Fanuc TP program (LS listing): FM194002.ls

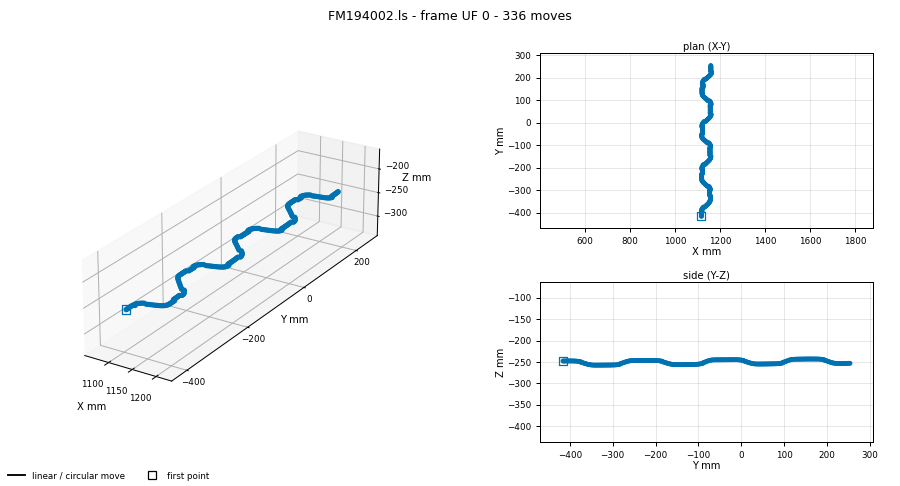
[picture p0: tool path of FM194002.ls in frame UF 0, 336 of 336 moves have a stored position in this frame; points joined in program order, loops and branches not executed]
/PROG  FM194002
/ATTR
OWNER		= MNEDITOR;
COMMENT		= "Auto FANUC move";
PROG_SIZE	= 0;
CREATE		= DATE 26-04-24  TIME 19:40:02;
MODIFIED	= DATE 26-04-24  TIME 19:40:02;
FILE_NAME	= ;
VERSION		= 0;
LINE_COUNT	= 341;
MEMORY_SIZE	= 0;
PROTECT		= READ_WRITE;
TCD:  STACK_SIZE	= 0,
      TASK_PRIORITY	= 50,
      TIME_SLICE	= 0,
      BUSY_LAMP_OFF	= 0,
      ABORT_REQUEST	= 0,
      PAUSE_REQUEST	= 0;
DEFAULT_GROUP	= 1,*,*,*,*;
CONTROL_CODE	= 00000000 00000000;
/MN
   1:  UFRAME_NUM=0 ;
   2:  UTOOL_NUM=1 ;
   3:  R[93]=10 ;
   4:  L P[1] 7mm/sec FINE ;
   5:  L P[2] 7mm/sec FINE ;
   6:  L P[3] 7mm/sec FINE ;
   7:  L P[4] 7mm/sec FINE ;
   8:  L P[5] 7mm/sec FINE ;
   9:  L P[6] 7mm/sec FINE ;
  10:  L P[7] 7mm/sec FINE ;
  11:  L P[8] 7mm/sec FINE ;
  12:  L P[9] 7mm/sec FINE ;
  13:  L P[10] 7mm/sec FINE ;
  14:  L P[11] 7mm/sec FINE ;
  15:  L P[12] 7mm/sec FINE ;
  16:  L P[13] 7mm/sec FINE ;
  17:  L P[14] 7mm/sec FINE ;
  18:  L P[15] 7mm/sec FINE ;
  19:  L P[16] 7mm/sec FINE ;
  20:  L P[17] 7mm/sec FINE ;
  21:  L P[18] 7mm/sec FINE ;
  22:  L P[19] 7mm/sec FINE ;
  23:  L P[20] 7mm/sec FINE ;
  24:  L P[21] 7mm/sec FINE ;
  25:  L P[22] 7mm/sec FINE ;
  26:  L P[23] 7mm/sec FINE ;
  27:  L P[24] 7mm/sec FINE ;
  28:  L P[25] 7mm/sec FINE ;
  29:  L P[26] 7mm/sec FINE ;
  30:  L P[27] 7mm/sec FINE ;
  31:  L P[28] 7mm/sec FINE ;
  32:  L P[29] 7mm/sec FINE ;
  33:  L P[30] 7mm/sec FINE ;
  34:  L P[31] 7mm/sec FINE ;
  35:  L P[32] 7mm/sec FINE ;
  36:  L P[33] 7mm/sec FINE ;
  37:  L P[34] 7mm/sec FINE ;
  38:  L P[35] 7mm/sec FINE ;
  39:  L P[36] 7mm/sec FINE ;
  40:  L P[37] 7mm/sec FINE ;
  41:  L P[38] 7mm/sec FINE ;
  42:  L P[39] 7mm/sec FINE ;
  43:  L P[40] 7mm/sec FINE ;
  44:  L P[41] 7mm/sec FINE ;
  45:  L P[42] 7mm/sec FINE ;
  46:  L P[43] 7mm/sec FINE ;
  47:  L P[44] 7mm/sec FINE ;
  48:  L P[45] 7mm/sec FINE ;
  49:  L P[46] 7mm/sec FINE ;
  50:  L P[47] 7mm/sec FINE ;
  51:  L P[48] 7mm/sec FINE ;
  52:  L P[49] 7mm/sec FINE ;
  53:  L P[50] 7mm/sec FINE ;
  54:  L P[51] 7mm/sec FINE ;
  55:  L P[52] 7mm/sec FINE ;
  56:  L P[53] 7mm/sec FINE ;
  57:  L P[54] 7mm/sec FINE ;
  58:  L P[55] 7mm/sec FINE ;
  59:  L P[56] 7mm/sec FINE ;
  60:  L P[57] 7mm/sec FINE ;
  61:  L P[58] 7mm/sec FINE ;
  62:  L P[59] 7mm/sec FINE ;
  63:  L P[60] 7mm/sec FINE ;
  64:  L P[61] 7mm/sec FINE ;
  65:  L P[62] 7mm/sec FINE ;
  66:  L P[63] 7mm/sec FINE ;
  67:  L P[64] 7mm/sec FINE ;
  68:  L P[65] 7mm/sec FINE ;
  69:  L P[66] 7mm/sec FINE ;
  70:  L P[67] 7mm/sec FINE ;
  71:  L P[68] 7mm/sec FINE ;
  72:  L P[69] 7mm/sec FINE ;
  73:  L P[70] 7mm/sec FINE ;
  74:  L P[71] 7mm/sec FINE ;
  75:  L P[72] 7mm/sec FINE ;
  76:  L P[73] 7mm/sec FINE ;
  77:  L P[74] 7mm/sec FINE ;
  78:  L P[75] 7mm/sec FINE ;
  79:  L P[76] 7mm/sec FINE ;
  80:  L P[77] 7mm/sec FINE ;
  81:  L P[78] 7mm/sec FINE ;
  82:  L P[79] 7mm/sec FINE ;
  83:  L P[80] 7mm/sec FINE ;
  84:  L P[81] 7mm/sec FINE ;
  85:  L P[82] 7mm/sec FINE ;
  86:  L P[83] 7mm/sec FINE ;
  87:  L P[84] 7mm/sec FINE ;
  88:  L P[85] 7mm/sec FINE ;
  89:  L P[86] 7mm/sec FINE ;
  90:  L P[87] 7mm/sec FINE ;
  91:  L P[88] 7mm/sec FINE ;
  92:  L P[89] 7mm/sec FINE ;
  93:  L P[90] 7mm/sec FINE ;
  94:  L P[91] 7mm/sec FINE ;
  95:  L P[92] 7mm/sec FINE ;
  96:  L P[93] 7mm/sec FINE ;
  97:  L P[94] 7mm/sec FINE ;
  98:  L P[95] 7mm/sec FINE ;
  99:  L P[96] 7mm/sec FINE ;
 100:  L P[97] 7mm/sec FINE ;
 101:  L P[98] 7mm/sec FINE ;
 102:  L P[99] 7mm/sec FINE ;
 103:  L P[100] 7mm/sec FINE ;
 104:  L P[101] 7mm/sec FINE ;
 105:  L P[102] 7mm/sec FINE ;
 106:  L P[103] 7mm/sec FINE ;
 107:  L P[104] 7mm/sec FINE ;
 108:  L P[105] 7mm/sec FINE ;
 109:  L P[106] 7mm/sec FINE ;
 110:  L P[107] 7mm/sec FINE ;
 111:  L P[108] 7mm/sec FINE ;
 112:  L P[109] 7mm/sec FINE ;
 113:  L P[110] 7mm/sec FINE ;
 114:  L P[111] 7mm/sec FINE ;
 115:  L P[112] 7mm/sec FINE ;
 116:  L P[113] 7mm/sec FINE ;
 117:  L P[114] 7mm/sec FINE ;
 118:  L P[115] 7mm/sec FINE ;
 119:  L P[116] 7mm/sec FINE ;
 120:  L P[117] 7mm/sec FINE ;
 121:  L P[118] 7mm/sec FINE ;
 122:  L P[119] 7mm/sec FINE ;
 123:  L P[120] 7mm/sec FINE ;
 124:  L P[121] 7mm/sec FINE ;
 125:  L P[122] 7mm/sec FINE ;
 126:  L P[123] 7mm/sec FINE ;
 127:  L P[124] 7mm/sec FINE ;
 128:  L P[125] 7mm/sec FINE ;
 129:  L P[126] 7mm/sec FINE ;
 130:  L P[127] 7mm/sec FINE ;
 131:  L P[128] 7mm/sec FINE ;
 132:  L P[129] 7mm/sec FINE ;
 133:  L P[130] 7mm/sec FINE ;
 134:  L P[131] 7mm/sec FINE ;
 135:  L P[132] 7mm/sec FINE ;
 136:  L P[133] 7mm/sec FINE ;
 137:  L P[134] 7mm/sec FINE ;
 138:  L P[135] 7mm/sec FINE ;
 139:  L P[136] 7mm/sec FINE ;
 140:  L P[137] 7mm/sec FINE ;
 141:  L P[138] 7mm/sec FINE ;
 142:  L P[139] 7mm/sec FINE ;
 143:  L P[140] 7mm/sec FINE ;
 144:  L P[141] 7mm/sec FINE ;
 145:  L P[142] 7mm/sec FINE ;
 146:  L P[143] 7mm/sec FINE ;
 147:  L P[144] 7mm/sec FINE ;
 148:  L P[145] 7mm/sec FINE ;
 149:  L P[146] 7mm/sec FINE ;
 150:  L P[147] 7mm/sec FINE ;
 151:  L P[148] 7mm/sec FINE ;
 152:  L P[149] 7mm/sec FINE ;
 153:  L P[150] 7mm/sec FINE ;
 154:  L P[151] 7mm/sec FINE ;
 155:  L P[152] 7mm/sec FINE ;
 156:  L P[153] 7mm/sec FINE ;
 157:  L P[154] 7mm/sec FINE ;
 158:  L P[155] 7mm/sec FINE ;
 159:  L P[156] 7mm/sec FINE ;
 160:  L P[157] 7mm/sec FINE ;
 161:  L P[158] 7mm/sec FINE ;
 162:  L P[159] 7mm/sec FINE ;
 163:  L P[160] 7mm/sec FINE ;
 164:  L P[161] 7mm/sec FINE ;
 165:  L P[162] 7mm/sec FINE ;
 166:  L P[163] 7mm/sec FINE ;
 167:  L P[164] 7mm/sec FINE ;
 168:  L P[165] 7mm/sec FINE ;
 169:  L P[166] 7mm/sec FINE ;
 170:  L P[167] 7mm/sec FINE ;
 171:  L P[168] 7mm/sec FINE ;
 172:  L P[169] 7mm/sec FINE ;
 173:  L P[170] 7mm/sec FINE ;
 174:  L P[171] 7mm/sec FINE ;
 175:  L P[172] 7mm/sec FINE ;
 176:  L P[173] 7mm/sec FINE ;
 177:  L P[174] 7mm/sec FINE ;
 178:  L P[175] 7mm/sec FINE ;
 179:  L P[176] 7mm/sec FINE ;
 180:  L P[177] 7mm/sec FINE ;
 181:  L P[178] 7mm/sec FINE ;
 182:  L P[179] 7mm/sec FINE ;
 183:  L P[180] 7mm/sec FINE ;
 184:  L P[181] 7mm/sec FINE ;
 185:  L P[182] 7mm/sec FINE ;
 186:  L P[183] 7mm/sec FINE ;
 187:  L P[184] 7mm/sec FINE ;
 188:  L P[185] 7mm/sec FINE ;
 189:  L P[186] 7mm/sec FINE ;
 190:  L P[187] 7mm/sec FINE ;
 191:  L P[188] 7mm/sec FINE ;
 192:  L P[189] 7mm/sec FINE ;
 193:  L P[190] 7mm/sec FINE ;
 194:  L P[191] 7mm/sec FINE ;
 195:  L P[192] 7mm/sec FINE ;
 196:  L P[193] 7mm/sec FINE ;
 197:  L P[194] 7mm/sec FINE ;
 198:  L P[195] 7mm/sec FINE ;
 199:  L P[196] 7mm/sec FINE ;
 200:  L P[197] 7mm/sec FINE ;
 201:  L P[198] 7mm/sec FINE ;
 202:  L P[199] 7mm/sec FINE ;
 203:  L P[200] 7mm/sec FINE ;
 204:  L P[201] 7mm/sec FINE ;
 205:  L P[202] 7mm/sec FINE ;
 206:  L P[203] 7mm/sec FINE ;
 207:  L P[204] 7mm/sec FINE ;
 208:  L P[205] 7mm/sec FINE ;
 209:  L P[206] 7mm/sec FINE ;
 210:  L P[207] 7mm/sec FINE ;
 211:  L P[208] 7mm/sec FINE ;
 212:  L P[209] 7mm/sec FINE ;
 213:  L P[210] 7mm/sec FINE ;
 214:  L P[211] 7mm/sec FINE ;
 215:  L P[212] 7mm/sec FINE ;
 216:  L P[213] 7mm/sec FINE ;
 217:  L P[214] 7mm/sec FINE ;
 218:  L P[215] 7mm/sec FINE ;
 219:  L P[216] 7mm/sec FINE ;
 220:  L P[217] 7mm/sec FINE ;
 221:  L P[218] 7mm/sec FINE ;
 222:  L P[219] 7mm/sec FINE ;
 223:  L P[220] 7mm/sec FINE ;
 224:  L P[221] 7mm/sec FINE ;
 225:  L P[222] 7mm/sec FINE ;
 226:  L P[223] 7mm/sec FINE ;
 227:  L P[224] 7mm/sec FINE ;
 228:  L P[225] 7mm/sec FINE ;
 229:  L P[226] 7mm/sec FINE ;
 230:  L P[227] 7mm/sec FINE ;
 231:  L P[228] 7mm/sec FINE ;
 232:  L P[229] 7mm/sec FINE ;
 233:  L P[230] 7mm/sec FINE ;
 234:  L P[231] 7mm/sec FINE ;
 235:  L P[232] 7mm/sec FINE ;
 236:  L P[233] 7mm/sec FINE ;
 237:  L P[234] 7mm/sec FINE ;
 238:  L P[235] 7mm/sec FINE ;
 239:  L P[236] 7mm/sec FINE ;
 240:  L P[237] 7mm/sec FINE ;
 241:  L P[238] 7mm/sec FINE ;
 242:  L P[239] 7mm/sec FINE ;
 243:  L P[240] 7mm/sec FINE ;
 244:  L P[241] 7mm/sec FINE ;
 245:  L P[242] 7mm/sec FINE ;
 246:  L P[243] 7mm/sec FINE ;
 247:  L P[244] 7mm/sec FINE ;
 248:  L P[245] 7mm/sec FINE ;
 249:  L P[246] 7mm/sec FINE ;
 250:  L P[247] 7mm/sec FINE ;
 251:  L P[248] 7mm/sec FINE ;
 252:  L P[249] 7mm/sec FINE ;
 253:  L P[250] 7mm/sec FINE ;
 254:  L P[251] 7mm/sec FINE ;
 255:  L P[252] 7mm/sec FINE ;
 256:  L P[253] 7mm/sec FINE ;
 257:  L P[254] 7mm/sec FINE ;
 258:  L P[255] 7mm/sec FINE ;
 259:  L P[256] 7mm/sec FINE ;
 260:  L P[257] 7mm/sec FINE ;
 261:  L P[258] 7mm/sec FINE ;
 262:  L P[259] 7mm/sec FINE ;
 263:  L P[260] 7mm/sec FINE ;
 264:  L P[261] 7mm/sec FINE ;
 265:  L P[262] 7mm/sec FINE ;
 266:  L P[263] 7mm/sec FINE ;
 267:  L P[264] 7mm/sec FINE ;
 268:  L P[265] 7mm/sec FINE ;
 269:  L P[266] 7mm/sec FINE ;
 270:  L P[267] 7mm/sec FINE ;
 271:  L P[268] 7mm/sec FINE ;
 272:  L P[269] 7mm/sec FINE ;
 273:  L P[270] 7mm/sec FINE ;
 274:  L P[271] 7mm/sec FINE ;
 275:  L P[272] 7mm/sec FINE ;
 276:  L P[273] 7mm/sec FINE ;
 277:  L P[274] 7mm/sec FINE ;
 278:  L P[275] 7mm/sec FINE ;
 279:  L P[276] 7mm/sec FINE ;
 280:  L P[277] 7mm/sec FINE ;
 281:  L P[278] 7mm/sec FINE ;
 282:  L P[279] 7mm/sec FINE ;
 283:  L P[280] 7mm/sec FINE ;
 284:  L P[281] 7mm/sec FINE ;
 285:  L P[282] 7mm/sec FINE ;
 286:  L P[283] 7mm/sec FINE ;
 287:  L P[284] 7mm/sec FINE ;
 288:  L P[285] 7mm/sec FINE ;
 289:  L P[286] 7mm/sec FINE ;
 290:  L P[287] 7mm/sec FINE ;
 291:  L P[288] 7mm/sec FINE ;
 292:  L P[289] 7mm/sec FINE ;
 293:  L P[290] 7mm/sec FINE ;
 294:  L P[291] 7mm/sec FINE ;
 295:  L P[292] 7mm/sec FINE ;
 296:  L P[293] 7mm/sec FINE ;
 297:  L P[294] 7mm/sec FINE ;
 298:  L P[295] 7mm/sec FINE ;
 299:  L P[296] 7mm/sec FINE ;
 300:  L P[297] 7mm/sec FINE ;
 301:  L P[298] 7mm/sec FINE ;
 302:  L P[299] 7mm/sec FINE ;
 303:  L P[300] 7mm/sec FINE ;
 304:  L P[301] 7mm/sec FINE ;
 305:  L P[302] 7mm/sec FINE ;
 306:  L P[303] 7mm/sec FINE ;
 307:  L P[304] 7mm/sec FINE ;
 308:  L P[305] 7mm/sec FINE ;
 309:  L P[306] 7mm/sec FINE ;
 310:  L P[307] 7mm/sec FINE ;
 311:  L P[308] 7mm/sec FINE ;
 312:  L P[309] 7mm/sec FINE ;
 313:  L P[310] 7mm/sec FINE ;
 314:  L P[311] 7mm/sec FINE ;
 315:  L P[312] 7mm/sec FINE ;
 316:  L P[313] 7mm/sec FINE ;
 317:  L P[314] 7mm/sec FINE ;
 318:  L P[315] 7mm/sec FINE ;
 319:  L P[316] 7mm/sec FINE ;
 320:  L P[317] 7mm/sec FINE ;
 321:  L P[318] 7mm/sec FINE ;
 322:  L P[319] 7mm/sec FINE ;
 323:  L P[320] 7mm/sec FINE ;
 324:  L P[321] 7mm/sec FINE ;
 325:  L P[322] 7mm/sec FINE ;
 326:  L P[323] 7mm/sec FINE ;
 327:  L P[324] 7mm/sec FINE ;
 328:  L P[325] 7mm/sec FINE ;
 329:  L P[326] 7mm/sec FINE ;
 330:  L P[327] 7mm/sec FINE ;
 331:  L P[328] 7mm/sec FINE ;
 332:  L P[329] 7mm/sec FINE ;
 333:  L P[330] 7mm/sec FINE ;
 334:  L P[331] 7mm/sec FINE ;
 335:  L P[332] 7mm/sec FINE ;
 336:  L P[333] 7mm/sec FINE ;
 337:  L P[334] 7mm/sec FINE ;
 338:  L P[335] 7mm/sec FINE ;
 339:  L P[336] 7mm/sec FINE ;
 340:  R[93]=1 ;
 341:  END ;
/POS
P[1]{
   GP1:
	UF : 0, UT : 1,		CONFIG : 'N U T, 0, 0, 0',
	X = 1117.903  mm,	Y = -416.081  mm,	Z = -247.708  mm,
	W = 0.000 deg,	P = 30.000 deg,	R = 175.406 deg
};
P[2]{
   GP1:
	UF : 0, UT : 1,		CONFIG : 'N U T, 0, 0, 0',
	X = 1117.822  mm,	Y = -414.081  mm,	Z = -247.687  mm,
	W = 0.000 deg,	P = 30.000 deg,	R = 175.406 deg
};
P[3]{
   GP1:
	UF : 0, UT : 1,		CONFIG : 'N U T, 0, 0, 0',
	X = 1117.741  mm,	Y = -412.076  mm,	Z = -247.659  mm,
	W = 0.000 deg,	P = 30.000 deg,	R = 175.406 deg
};
P[4]{
   GP1:
	UF : 0, UT : 1,		CONFIG : 'N U T, 0, 0, 0',
	X = 1117.669  mm,	Y = -410.061  mm,	Z = -247.629  mm,
	W = 0.000 deg,	P = 30.000 deg,	R = 175.406 deg
};
P[5]{
   GP1:
	UF : 0, UT : 1,		CONFIG : 'N U T, 0, 0, 0',
	X = 1117.617  mm,	Y = -408.050  mm,	Z = -247.600  mm,
	W = 0.000 deg,	P = 30.000 deg,	R = 175.406 deg
};
P[6]{
   GP1:
	UF : 0, UT : 1,		CONFIG : 'N U T, 0, 0, 0',
	X = 1117.569  mm,	Y = -406.040  mm,	Z = -247.570  mm,
	W = 0.000 deg,	P = 30.000 deg,	R = 175.406 deg
};
P[7]{
   GP1:
	UF : 0, UT : 1,		CONFIG : 'N U T, 0, 0, 0',
	X = 1117.536  mm,	Y = -404.021  mm,	Z = -247.543  mm,
	W = 0.000 deg,	P = 30.000 deg,	R = 175.406 deg
};
P[8]{
   GP1:
	UF : 0, UT : 1,		CONFIG : 'N U T, 0, 0, 0',
	X = 1117.527  mm,	Y = -402.002  mm,	Z = -247.518  mm,
	W = 0.000 deg,	P = 30.000 deg,	R = 175.406 deg
};
P[9]{
   GP1:
	UF : 0, UT : 1,		CONFIG : 'N U T, 0, 0, 0',
	X = 1117.533  mm,	Y = -399.972  mm,	Z = -247.500  mm,
	W = 0.000 deg,	P = 30.000 deg,	R = 175.406 deg
};
P[10]{
   GP1:
	UF : 0, UT : 1,		CONFIG : 'N U T, 0, 0, 0',
	X = 1117.583  mm,	Y = -397.934  mm,	Z = -247.497  mm,
	W = 0.000 deg,	P = 30.000 deg,	R = 175.406 deg
};
P[11]{
   GP1:
	UF : 0, UT : 1,		CONFIG : 'N U T, 0, 0, 0',
	X = 1117.668  mm,	Y = -395.878  mm,	Z = -247.506  mm,
	W = 0.000 deg,	P = 30.000 deg,	R = 175.406 deg
};
P[12]{
   GP1:
	UF : 0, UT : 1,		CONFIG : 'N U T, 0, 0, 0',
	X = 1121.814  mm,	Y = -394.222  mm,	Z = -247.528  mm,
	W = 0.000 deg,	P = 30.000 deg,	R = 175.406 deg
};
P[13]{
   GP1:
	UF : 0, UT : 1,		CONFIG : 'N U T, 0, 0, 0',
	X = 1118.142  mm,	Y = -391.652  mm,	Z = -247.591  mm,
	W = 0.000 deg,	P = 30.000 deg,	R = 169.886 deg
};
P[14]{
   GP1:
	UF : 0, UT : 1,		CONFIG : 'N U T, 0, 0, 0',
	X = 1118.595  mm,	Y = -389.505  mm,	Z = -247.675  mm,
	W = 0.000 deg,	P = 30.000 deg,	R = 162.214 deg
};
P[15]{
   GP1:
	UF : 0, UT : 1,		CONFIG : 'N U T, 0, 0, 0',
	X = 1119.241  mm,	Y = -387.351  mm,	Z = -247.801  mm,
	W = 0.000 deg,	P = 30.000 deg,	R = 154.369 deg
};
P[16]{
   GP1:
	UF : 0, UT : 1,		CONFIG : 'N U T, 0, 0, 0',
	X = 1120.076  mm,	Y = -385.192  mm,	Z = -247.960  mm,
	W = 0.000 deg,	P = 30.000 deg,	R = 146.306 deg
};
P[17]{
   GP1:
	UF : 0, UT : 1,		CONFIG : 'N U T, 0, 0, 0',
	X = 1121.155  mm,	Y = -383.023  mm,	Z = -248.138  mm,
	W = 0.000 deg,	P = 30.000 deg,	R = 137.902 deg
};
P[18]{
   GP1:
	UF : 0, UT : 1,		CONFIG : 'N U T, 0, 0, 0',
	X = 1122.476  mm,	Y = -380.896  mm,	Z = -248.389  mm,
	W = 0.000 deg,	P = 30.000 deg,	R = 137.902 deg
};
P[19]{
   GP1:
	UF : 0, UT : 1,		CONFIG : 'N U T, 0, 0, 0',
	X = 1123.929  mm,	Y = -378.824  mm,	Z = -248.707  mm,
	W = 0.000 deg,	P = 30.000 deg,	R = 137.902 deg
};
P[20]{
   GP1:
	UF : 0, UT : 1,		CONFIG : 'N U T, 0, 0, 0',
	X = 1125.487  mm,	Y = -376.754  mm,	Z = -249.062  mm,
	W = 0.000 deg,	P = 30.000 deg,	R = 137.902 deg
};
P[21]{
   GP1:
	UF : 0, UT : 1,		CONFIG : 'N U T, 0, 0, 0',
	X = 1127.242  mm,	Y = -374.667  mm,	Z = -249.504  mm,
	W = 0.000 deg,	P = 30.000 deg,	R = 137.902 deg
};
P[22]{
   GP1:
	UF : 0, UT : 1,		CONFIG : 'N U T, 0, 0, 0',
	X = 1132.067  mm,	Y = -375.388  mm,	Z = -250.027  mm,
	W = 0.000 deg,	P = 30.000 deg,	R = 137.902 deg
};
P[23]{
   GP1:
	UF : 0, UT : 1,		CONFIG : 'N U T, 0, 0, 0',
	X = 1134.024  mm,	Y = -373.390  mm,	Z = -250.598  mm,
	W = 0.000 deg,	P = 30.000 deg,	R = 137.902 deg
};
P[24]{
   GP1:
	UF : 0, UT : 1,		CONFIG : 'N U T, 0, 0, 0',
	X = 1135.917  mm,	Y = -371.406  mm,	Z = -251.204  mm,
	W = 0.000 deg,	P = 30.000 deg,	R = 137.902 deg
};
P[25]{
   GP1:
	UF : 0, UT : 1,		CONFIG : 'N U T, 0, 0, 0',
	X = 1137.928  mm,	Y = -369.443  mm,	Z = -251.855  mm,
	W = 0.000 deg,	P = 30.000 deg,	R = 137.902 deg
};
P[26]{
   GP1:
	UF : 0, UT : 1,		CONFIG : 'N U T, 0, 0, 0',
	X = 1140.023  mm,	Y = -367.467  mm,	Z = -252.522  mm,
	W = 0.000 deg,	P = 30.000 deg,	R = 137.902 deg
};
P[27]{
   GP1:
	UF : 0, UT : 1,		CONFIG : 'N U T, 0, 0, 0',
	X = 1142.218  mm,	Y = -365.469  mm,	Z = -253.201  mm,
	W = 0.000 deg,	P = 30.000 deg,	R = 137.902 deg
};
P[28]{
   GP1:
	UF : 0, UT : 1,		CONFIG : 'N U T, 0, 0, 0',
	X = 1144.405  mm,	Y = -363.418  mm,	Z = -253.848  mm,
	W = 0.000 deg,	P = 30.000 deg,	R = 137.902 deg
};
P[29]{
   GP1:
	UF : 0, UT : 1,		CONFIG : 'N U T, 0, 0, 0',
	X = 1146.326  mm,	Y = -361.385  mm,	Z = -254.414  mm,
	W = 0.000 deg,	P = 30.000 deg,	R = 137.902 deg
};
P[30]{
   GP1:
	UF : 0, UT : 1,		CONFIG : 'N U T, 0, 0, 0',
	X = 1148.257  mm,	Y = -359.405  mm,	Z = -254.982  mm,
	W = 0.000 deg,	P = 30.000 deg,	R = 146.247 deg
};
P[31]{
   GP1:
	UF : 0, UT : 1,		CONFIG : 'N U T, 0, 0, 0',
	X = 1150.309  mm,	Y = -357.349  mm,	Z = -255.565  mm,
	W = 0.000 deg,	P = 30.000 deg,	R = 158.379 deg
};
P[32]{
   GP1:
	UF : 0, UT : 1,		CONFIG : 'N U T, 0, 0, 0',
	X = 1152.072  mm,	Y = -355.220  mm,	Z = -256.043  mm,
	W = 0.000 deg,	P = 30.000 deg,	R = 169.473 deg
};
P[33]{
   GP1:
	UF : 0, UT : 1,		CONFIG : 'N U T, 0, 0, 0',
	X = 1153.595  mm,	Y = -353.081  mm,	Z = -256.439  mm,
	W = 0.000 deg,	P = 30.000 deg,	R = 179.925 deg
};
P[34]{
   GP1:
	UF : 0, UT : 1,		CONFIG : 'N U T, 0, 0, 0',
	X = 1154.836  mm,	Y = -350.912  mm,	Z = -256.747  mm,
	W = 0.000 deg,	P = 30.000 deg,	R = 179.925 deg
};
P[35]{
   GP1:
	UF : 0, UT : 1,		CONFIG : 'N U T, 0, 0, 0',
	X = 1155.808  mm,	Y = -348.771  mm,	Z = -256.977  mm,
	W = 0.000 deg,	P = 30.000 deg,	R = 179.925 deg
};
P[36]{
   GP1:
	UF : 0, UT : 1,		CONFIG : 'N U T, 0, 0, 0',
	X = 1156.640  mm,	Y = -346.586  mm,	Z = -257.166  mm,
	W = 0.000 deg,	P = 30.000 deg,	R = 179.925 deg
};
P[37]{
   GP1:
	UF : 0, UT : 1,		CONFIG : 'N U T, 0, 0, 0',
	X = 1157.161  mm,	Y = -344.331  mm,	Z = -257.271  mm,
	W = 0.000 deg,	P = 30.000 deg,	R = 179.925 deg
};
P[38]{
   GP1:
	UF : 0, UT : 1,		CONFIG : 'N U T, 0, 0, 0',
	X = 1157.393  mm,	Y = -342.172  mm,	Z = -257.304  mm,
	W = 0.000 deg,	P = 30.000 deg,	R = 179.925 deg
};
P[39]{
   GP1:
	UF : 0, UT : 1,		CONFIG : 'N U T, 0, 0, 0',
	X = 1157.531  mm,	Y = -340.095  mm,	Z = -257.316  mm,
	W = 0.000 deg,	P = 30.000 deg,	R = 179.925 deg
};
P[40]{
   GP1:
	UF : 0, UT : 1,		CONFIG : 'N U T, 0, 0, 0',
	X = 1157.590  mm,	Y = -338.047  mm,	Z = -257.316  mm,
	W = 0.000 deg,	P = 30.000 deg,	R = 179.925 deg
};
P[41]{
   GP1:
	UF : 0, UT : 1,		CONFIG : 'N U T, 0, 0, 0',
	X = 1157.627  mm,	Y = -336.032  mm,	Z = -257.313  mm,
	W = 0.000 deg,	P = 30.000 deg,	R = 179.925 deg
};
P[42]{
   GP1:
	UF : 0, UT : 1,		CONFIG : 'N U T, 0, 0, 0',
	X = 1157.653  mm,	Y = -334.022  mm,	Z = -257.307  mm,
	W = 0.000 deg,	P = 30.000 deg,	R = 179.925 deg
};
P[43]{
   GP1:
	UF : 0, UT : 1,		CONFIG : 'N U T, 0, 0, 0',
	X = 1157.672  mm,	Y = -332.016  mm,	Z = -257.298  mm,
	W = 0.000 deg,	P = 30.000 deg,	R = 179.925 deg
};
P[44]{
   GP1:
	UF : 0, UT : 1,		CONFIG : 'N U T, 0, 0, 0',
	X = 1157.685  mm,	Y = -330.011  mm,	Z = -257.283  mm,
	W = 0.000 deg,	P = 30.000 deg,	R = 179.925 deg
};
P[45]{
   GP1:
	UF : 0, UT : 1,		CONFIG : 'N U T, 0, 0, 0',
	X = 1157.693  mm,	Y = -328.007  mm,	Z = -257.262  mm,
	W = 0.000 deg,	P = 30.000 deg,	R = 179.925 deg
};
P[46]{
   GP1:
	UF : 0, UT : 1,		CONFIG : 'N U T, 0, 0, 0',
	X = 1157.700  mm,	Y = -326.005  mm,	Z = -257.241  mm,
	W = 0.000 deg,	P = 30.000 deg,	R = 179.925 deg
};
P[47]{
   GP1:
	UF : 0, UT : 1,		CONFIG : 'N U T, 0, 0, 0',
	X = 1157.703  mm,	Y = -324.003  mm,	Z = -257.219  mm,
	W = 0.000 deg,	P = 30.000 deg,	R = 179.925 deg
};
P[48]{
   GP1:
	UF : 0, UT : 1,		CONFIG : 'N U T, 0, 0, 0',
	X = 1153.706  mm,	Y = -321.999  mm,	Z = -257.197  mm,
	W = 0.000 deg,	P = 30.000 deg,	R = 179.925 deg
};
P[49]{
   GP1:
	UF : 0, UT : 1,		CONFIG : 'N U T, 0, 0, 0',
	X = 1153.704  mm,	Y = -320.005  mm,	Z = -257.178  mm,
	W = 0.000 deg,	P = 30.000 deg,	R = 179.925 deg
};
P[50]{
   GP1:
	UF : 0, UT : 1,		CONFIG : 'N U T, 0, 0, 0',
	X = 1153.696  mm,	Y = -318.010  mm,	Z = -257.160  mm,
	W = 0.000 deg,	P = 30.000 deg,	R = 179.925 deg
};
P[51]{
   GP1:
	UF : 0, UT : 1,		CONFIG : 'N U T, 0, 0, 0',
	X = 1153.685  mm,	Y = -316.013  mm,	Z = -257.148  mm,
	W = 0.000 deg,	P = 30.000 deg,	R = 179.925 deg
};
P[52]{
   GP1:
	UF : 0, UT : 1,		CONFIG : 'N U T, 0, 0, 0',
	X = 1153.670  mm,	Y = -314.020  mm,	Z = -257.138  mm,
	W = 0.000 deg,	P = 30.000 deg,	R = 179.925 deg
};
P[53]{
   GP1:
	UF : 0, UT : 1,		CONFIG : 'N U T, 0, 0, 0',
	X = 1153.645  mm,	Y = -312.032  mm,	Z = -257.126  mm,
	W = 0.000 deg,	P = 30.000 deg,	R = 179.925 deg
};
P[54]{
   GP1:
	UF : 0, UT : 1,		CONFIG : 'N U T, 0, 0, 0',
	X = 1153.607  mm,	Y = -310.048  mm,	Z = -257.109  mm,
	W = 0.000 deg,	P = 30.000 deg,	R = 179.925 deg
};
P[55]{
   GP1:
	UF : 0, UT : 1,		CONFIG : 'N U T, 0, 0, 0',
	X = 1153.548  mm,	Y = -308.060  mm,	Z = -257.085  mm,
	W = 0.000 deg,	P = 30.000 deg,	R = 179.925 deg
};
P[56]{
   GP1:
	UF : 0, UT : 1,		CONFIG : 'N U T, 0, 0, 0',
	X = 1153.487  mm,	Y = -306.064  mm,	Z = -257.061  mm,
	W = 0.000 deg,	P = 30.000 deg,	R = 179.925 deg
};
P[57]{
   GP1:
	UF : 0, UT : 1,		CONFIG : 'N U T, 0, 0, 0',
	X = 1153.420  mm,	Y = -304.075  mm,	Z = -257.035  mm,
	W = 0.000 deg,	P = 30.000 deg,	R = 179.925 deg
};
P[58]{
   GP1:
	UF : 0, UT : 1,		CONFIG : 'N U T, 0, 0, 0',
	X = 1153.338  mm,	Y = -302.094  mm,	Z = -257.001  mm,
	W = 0.000 deg,	P = 30.000 deg,	R = 179.925 deg
};
P[59]{
   GP1:
	UF : 0, UT : 1,		CONFIG : 'N U T, 0, 0, 0',
	X = 1157.227  mm,	Y = -299.889  mm,	Z = -256.960  mm,
	W = 0.000 deg,	P = 30.000 deg,	R = -172.261 deg
};
P[60]{
   GP1:
	UF : 0, UT : 1,		CONFIG : 'N U T, 0, 0, 0',
	X = 1157.108  mm,	Y = -297.863  mm,	Z = -256.914  mm,
	W = 0.000 deg,	P = 30.000 deg,	R = -163.648 deg
};
P[61]{
   GP1:
	UF : 0, UT : 1,		CONFIG : 'N U T, 0, 0, 0',
	X = 1156.941  mm,	Y = -295.770  mm,	Z = -256.860  mm,
	W = 0.000 deg,	P = 30.000 deg,	R = -155.021 deg
};
P[62]{
   GP1:
	UF : 0, UT : 1,		CONFIG : 'N U T, 0, 0, 0',
	X = 1156.585  mm,	Y = -293.494  mm,	Z = -256.766  mm,
	W = 0.000 deg,	P = 30.000 deg,	R = -146.317 deg
};
P[63]{
   GP1:
	UF : 0, UT : 1,		CONFIG : 'N U T, 0, 0, 0',
	X = 1155.778  mm,	Y = -291.291  mm,	Z = -256.533  mm,
	W = 0.000 deg,	P = 30.000 deg,	R = -137.092 deg
};
P[64]{
   GP1:
	UF : 0, UT : 1,		CONFIG : 'N U T, 0, 0, 0',
	X = 1154.940  mm,	Y = -289.140  mm,	Z = -256.291  mm,
	W = 0.000 deg,	P = 30.000 deg,	R = -137.092 deg
};
P[65]{
   GP1:
	UF : 0, UT : 1,		CONFIG : 'N U T, 0, 0, 0',
	X = 1153.690  mm,	Y = -286.928  mm,	Z = -255.943  mm,
	W = 0.000 deg,	P = 30.000 deg,	R = -137.092 deg
};
P[66]{
   GP1:
	UF : 0, UT : 1,		CONFIG : 'N U T, 0, 0, 0',
	X = 1152.204  mm,	Y = -284.813  mm,	Z = -255.513  mm,
	W = 0.000 deg,	P = 30.000 deg,	R = -137.092 deg
};
P[67]{
   GP1:
	UF : 0, UT : 1,		CONFIG : 'N U T, 0, 0, 0',
	X = 1150.545  mm,	Y = -282.671  mm,	Z = -255.041  mm,
	W = 0.000 deg,	P = 30.000 deg,	R = -137.092 deg
};
P[68]{
   GP1:
	UF : 0, UT : 1,		CONFIG : 'N U T, 0, 0, 0',
	X = 1145.642  mm,	Y = -283.430  mm,	Z = -254.415  mm,
	W = 0.000 deg,	P = 30.000 deg,	R = -137.092 deg
};
P[69]{
   GP1:
	UF : 0, UT : 1,		CONFIG : 'N U T, 0, 0, 0',
	X = 1143.569  mm,	Y = -281.439  mm,	Z = -253.764  mm,
	W = 0.000 deg,	P = 30.000 deg,	R = -137.092 deg
};
P[70]{
   GP1:
	UF : 0, UT : 1,		CONFIG : 'N U T, 0, 0, 0',
	X = 1141.558  mm,	Y = -279.486  mm,	Z = -253.115  mm,
	W = 0.000 deg,	P = 30.000 deg,	R = -137.092 deg
};
P[71]{
   GP1:
	UF : 0, UT : 1,		CONFIG : 'N U T, 0, 0, 0',
	X = 1139.168  mm,	Y = -277.477  mm,	Z = -252.354  mm,
	W = 0.000 deg,	P = 30.000 deg,	R = -137.092 deg
};
P[72]{
   GP1:
	UF : 0, UT : 1,		CONFIG : 'N U T, 0, 0, 0',
	X = 1137.118  mm,	Y = -275.431  mm,	Z = -251.708  mm,
	W = 0.000 deg,	P = 30.000 deg,	R = -137.092 deg
};
P[73]{
   GP1:
	UF : 0, UT : 1,		CONFIG : 'N U T, 0, 0, 0',
	X = 1135.038  mm,	Y = -273.445  mm,	Z = -251.008  mm,
	W = 0.000 deg,	P = 30.000 deg,	R = -137.092 deg
};
P[74]{
   GP1:
	UF : 0, UT : 1,		CONFIG : 'N U T, 0, 0, 0',
	X = 1132.925  mm,	Y = -271.417  mm,	Z = -250.292  mm,
	W = 0.000 deg,	P = 30.000 deg,	R = -137.092 deg
};
P[75]{
   GP1:
	UF : 0, UT : 1,		CONFIG : 'N U T, 0, 0, 0',
	X = 1131.034  mm,	Y = -269.457  mm,	Z = -249.652  mm,
	W = 0.000 deg,	P = 30.000 deg,	R = -137.092 deg
};
P[76]{
   GP1:
	UF : 0, UT : 1,		CONFIG : 'N U T, 0, 0, 0',
	X = 1128.718  mm,	Y = -267.465  mm,	Z = -248.952  mm,
	W = 0.000 deg,	P = 30.000 deg,	R = -144.940 deg
};
P[77]{
   GP1:
	UF : 0, UT : 1,		CONFIG : 'N U T, 0, 0, 0',
	X = 1126.623  mm,	Y = -265.346  mm,	Z = -248.378  mm,
	W = 0.000 deg,	P = 30.000 deg,	R = -157.359 deg
};
P[78]{
   GP1:
	UF : 0, UT : 1,		CONFIG : 'N U T, 0, 0, 0',
	X = 1124.911  mm,	Y = -263.289  mm,	Z = -247.921  mm,
	W = 0.000 deg,	P = 30.000 deg,	R = -168.781 deg
};
P[79]{
   GP1:
	UF : 0, UT : 1,		CONFIG : 'N U T, 0, 0, 0',
	X = 1123.138  mm,	Y = -261.212  mm,	Z = -247.447  mm,
	W = 0.000 deg,	P = 30.000 deg,	R = 179.652 deg
};
P[80]{
   GP1:
	UF : 0, UT : 1,		CONFIG : 'N U T, 0, 0, 0',
	X = 1121.702  mm,	Y = -259.072  mm,	Z = -247.117  mm,
	W = 0.000 deg,	P = 30.000 deg,	R = 179.652 deg
};
P[81]{
   GP1:
	UF : 0, UT : 1,		CONFIG : 'N U T, 0, 0, 0',
	X = 1120.407  mm,	Y = -256.906  mm,	Z = -246.842  mm,
	W = 0.000 deg,	P = 30.000 deg,	R = 179.652 deg
};
P[82]{
   GP1:
	UF : 0, UT : 1,		CONFIG : 'N U T, 0, 0, 0',
	X = 1119.423  mm,	Y = -254.501  mm,	Z = -246.659  mm,
	W = 0.000 deg,	P = 30.000 deg,	R = 179.652 deg
};
P[83]{
   GP1:
	UF : 0, UT : 1,		CONFIG : 'N U T, 0, 0, 0',
	X = 1119.162  mm,	Y = -252.164  mm,	Z = -246.603  mm,
	W = 0.000 deg,	P = 30.000 deg,	R = 179.652 deg
};
P[84]{
   GP1:
	UF : 0, UT : 1,		CONFIG : 'N U T, 0, 0, 0',
	X = 1119.033  mm,	Y = -250.103  mm,	Z = -246.560  mm,
	W = 0.000 deg,	P = 30.000 deg,	R = 179.652 deg
};
P[85]{
   GP1:
	UF : 0, UT : 1,		CONFIG : 'N U T, 0, 0, 0',
	X = 1118.950  mm,	Y = -248.057  mm,	Z = -246.519  mm,
	W = 0.000 deg,	P = 30.000 deg,	R = 179.652 deg
};
P[86]{
   GP1:
	UF : 0, UT : 1,		CONFIG : 'N U T, 0, 0, 0',
	X = 1118.916  mm,	Y = -246.021  mm,	Z = -246.492  mm,
	W = 0.000 deg,	P = 30.000 deg,	R = 179.652 deg
};
P[87]{
   GP1:
	UF : 0, UT : 1,		CONFIG : 'N U T, 0, 0, 0',
	X = 1118.906  mm,	Y = -244.003  mm,	Z = -246.468  mm,
	W = 0.000 deg,	P = 30.000 deg,	R = 179.652 deg
};
P[88]{
   GP1:
	UF : 0, UT : 1,		CONFIG : 'N U T, 0, 0, 0',
	X = 1118.910  mm,	Y = -241.997  mm,	Z = -246.451  mm,
	W = 0.000 deg,	P = 30.000 deg,	R = 179.652 deg
};
P[89]{
   GP1:
	UF : 0, UT : 1,		CONFIG : 'N U T, 0, 0, 0',
	X = 1118.913  mm,	Y = -239.996  mm,	Z = -246.434  mm,
	W = 0.000 deg,	P = 30.000 deg,	R = 179.652 deg
};
P[90]{
   GP1:
	UF : 0, UT : 1,		CONFIG : 'N U T, 0, 0, 0',
	X = 1118.917  mm,	Y = -237.995  mm,	Z = -246.415  mm,
	W = 0.000 deg,	P = 30.000 deg,	R = 179.652 deg
};
P[91]{
   GP1:
	UF : 0, UT : 1,		CONFIG : 'N U T, 0, 0, 0',
	X = 1118.923  mm,	Y = -235.994  mm,	Z = -246.394  mm,
	W = 0.000 deg,	P = 30.000 deg,	R = 179.652 deg
};
P[92]{
   GP1:
	UF : 0, UT : 1,		CONFIG : 'N U T, 0, 0, 0',
	X = 1118.929  mm,	Y = -233.993  mm,	Z = -246.378  mm,
	W = 0.000 deg,	P = 30.000 deg,	R = 179.652 deg
};
P[93]{
   GP1:
	UF : 0, UT : 1,		CONFIG : 'N U T, 0, 0, 0',
	X = 1118.936  mm,	Y = -231.993  mm,	Z = -246.364  mm,
	W = 0.000 deg,	P = 30.000 deg,	R = 179.652 deg
};
P[94]{
   GP1:
	UF : 0, UT : 1,		CONFIG : 'N U T, 0, 0, 0',
	X = 1118.942  mm,	Y = -229.994  mm,	Z = -246.348  mm,
	W = 0.000 deg,	P = 30.000 deg,	R = 179.652 deg
};
P[95]{
   GP1:
	UF : 0, UT : 1,		CONFIG : 'N U T, 0, 0, 0',
	X = 1118.948  mm,	Y = -227.990  mm,	Z = -246.333  mm,
	W = 0.000 deg,	P = 30.000 deg,	R = 179.652 deg
};
P[96]{
   GP1:
	UF : 0, UT : 1,		CONFIG : 'N U T, 0, 0, 0',
	X = 1122.962  mm,	Y = -226.020  mm,	Z = -246.316  mm,
	W = 0.000 deg,	P = 30.000 deg,	R = 179.652 deg
};
P[97]{
   GP1:
	UF : 0, UT : 1,		CONFIG : 'N U T, 0, 0, 0',
	X = 1122.987  mm,	Y = -224.026  mm,	Z = -246.304  mm,
	W = 0.000 deg,	P = 30.000 deg,	R = 179.652 deg
};
P[98]{
   GP1:
	UF : 0, UT : 1,		CONFIG : 'N U T, 0, 0, 0',
	X = 1123.014  mm,	Y = -222.030  mm,	Z = -246.293  mm,
	W = 0.000 deg,	P = 30.000 deg,	R = 179.652 deg
};
P[99]{
   GP1:
	UF : 0, UT : 1,		CONFIG : 'N U T, 0, 0, 0',
	X = 1123.048  mm,	Y = -220.037  mm,	Z = -246.280  mm,
	W = 0.000 deg,	P = 30.000 deg,	R = 179.652 deg
};
P[100]{
   GP1:
	UF : 0, UT : 1,		CONFIG : 'N U T, 0, 0, 0',
	X = 1123.088  mm,	Y = -218.051  mm,	Z = -246.267  mm,
	W = 0.000 deg,	P = 30.000 deg,	R = 179.652 deg
};
P[101]{
   GP1:
	UF : 0, UT : 1,		CONFIG : 'N U T, 0, 0, 0',
	X = 1123.149  mm,	Y = -216.067  mm,	Z = -246.260  mm,
	W = 0.000 deg,	P = 30.000 deg,	R = 179.652 deg
};
P[102]{
   GP1:
	UF : 0, UT : 1,		CONFIG : 'N U T, 0, 0, 0',
	X = 1123.221  mm,	Y = -214.068  mm,	Z = -246.254  mm,
	W = 0.000 deg,	P = 30.000 deg,	R = 179.652 deg
};
P[103]{
   GP1:
	UF : 0, UT : 1,		CONFIG : 'N U T, 0, 0, 0',
	X = 1123.286  mm,	Y = -212.068  mm,	Z = -246.255  mm,
	W = 0.000 deg,	P = 30.000 deg,	R = 179.652 deg
};
P[104]{
   GP1:
	UF : 0, UT : 1,		CONFIG : 'N U T, 0, 0, 0',
	X = 1123.357  mm,	Y = -210.081  mm,	Z = -246.257  mm,
	W = 0.000 deg,	P = 30.000 deg,	R = 179.652 deg
};
P[105]{
   GP1:
	UF : 0, UT : 1,		CONFIG : 'N U T, 0, 0, 0',
	X = 1123.447  mm,	Y = -208.107  mm,	Z = -246.265  mm,
	W = 0.000 deg,	P = 30.000 deg,	R = 179.652 deg
};
P[106]{
   GP1:
	UF : 0, UT : 1,		CONFIG : 'N U T, 0, 0, 0',
	X = 1119.579  mm,	Y = -205.848  mm,	Z = -246.280  mm,
	W = 0.000 deg,	P = 30.000 deg,	R = 172.109 deg
};
P[107]{
   GP1:
	UF : 0, UT : 1,		CONFIG : 'N U T, 0, 0, 0',
	X = 1119.767  mm,	Y = -203.777  mm,	Z = -246.306  mm,
	W = 0.000 deg,	P = 30.000 deg,	R = 163.850 deg
};
P[108]{
   GP1:
	UF : 0, UT : 1,		CONFIG : 'N U T, 0, 0, 0',
	X = 1120.055  mm,	Y = -201.642  mm,	Z = -246.357  mm,
	W = 0.000 deg,	P = 30.000 deg,	R = 155.549 deg
};
P[109]{
   GP1:
	UF : 0, UT : 1,		CONFIG : 'N U T, 0, 0, 0',
	X = 1120.547  mm,	Y = -199.499  mm,	Z = -246.457  mm,
	W = 0.000 deg,	P = 30.000 deg,	R = 147.099 deg
};
P[110]{
   GP1:
	UF : 0, UT : 1,		CONFIG : 'N U T, 0, 0, 0',
	X = 1121.153  mm,	Y = -197.389  mm,	Z = -246.574  mm,
	W = 0.000 deg,	P = 30.000 deg,	R = 138.529 deg
};
P[111]{
   GP1:
	UF : 0, UT : 1,		CONFIG : 'N U T, 0, 0, 0',
	X = 1121.912  mm,	Y = -195.252  mm,	Z = -246.733  mm,
	W = 0.000 deg,	P = 30.000 deg,	R = 138.529 deg
};
P[112]{
   GP1:
	UF : 0, UT : 1,		CONFIG : 'N U T, 0, 0, 0',
	X = 1122.893  mm,	Y = -193.083  mm,	Z = -246.935  mm,
	W = 0.000 deg,	P = 30.000 deg,	R = 138.529 deg
};
P[113]{
   GP1:
	UF : 0, UT : 1,		CONFIG : 'N U T, 0, 0, 0',
	X = 1124.136  mm,	Y = -190.935  mm,	Z = -247.164  mm,
	W = 0.000 deg,	P = 30.000 deg,	R = 138.529 deg
};
P[114]{
   GP1:
	UF : 0, UT : 1,		CONFIG : 'N U T, 0, 0, 0',
	X = 1125.568  mm,	Y = -188.827  mm,	Z = -247.478  mm,
	W = 0.000 deg,	P = 30.000 deg,	R = 138.529 deg
};
P[115]{
   GP1:
	UF : 0, UT : 1,		CONFIG : 'N U T, 0, 0, 0',
	X = 1127.155  mm,	Y = -186.762  mm,	Z = -247.866  mm,
	W = 0.000 deg,	P = 30.000 deg,	R = 138.529 deg
};
P[116]{
   GP1:
	UF : 0, UT : 1,		CONFIG : 'N U T, 0, 0, 0',
	X = 1128.829  mm,	Y = -184.689  mm,	Z = -248.300  mm,
	W = 0.000 deg,	P = 30.000 deg,	R = 138.529 deg
};
P[117]{
   GP1:
	UF : 0, UT : 1,		CONFIG : 'N U T, 0, 0, 0',
	X = 1133.651  mm,	Y = -185.373  mm,	Z = -248.827  mm,
	W = 0.000 deg,	P = 30.000 deg,	R = 138.529 deg
};
P[118]{
   GP1:
	UF : 0, UT : 1,		CONFIG : 'N U T, 0, 0, 0',
	X = 1135.538  mm,	Y = -183.405  mm,	Z = -249.377  mm,
	W = 0.000 deg,	P = 30.000 deg,	R = 138.529 deg
};
P[119]{
   GP1:
	UF : 0, UT : 1,		CONFIG : 'N U T, 0, 0, 0',
	X = 1137.539  mm,	Y = -181.436  mm,	Z = -249.975  mm,
	W = 0.000 deg,	P = 30.000 deg,	R = 138.529 deg
};
P[120]{
   GP1:
	UF : 0, UT : 1,		CONFIG : 'N U T, 0, 0, 0',
	X = 1139.635  mm,	Y = -179.435  mm,	Z = -250.657  mm,
	W = 0.000 deg,	P = 30.000 deg,	R = 138.529 deg
};
P[121]{
   GP1:
	UF : 0, UT : 1,		CONFIG : 'N U T, 0, 0, 0',
	X = 1141.666  mm,	Y = -177.427  mm,	Z = -251.292  mm,
	W = 0.000 deg,	P = 30.000 deg,	R = 138.529 deg
};
P[122]{
   GP1:
	UF : 0, UT : 1,		CONFIG : 'N U T, 0, 0, 0',
	X = 1143.712  mm,	Y = -175.434  mm,	Z = -251.920  mm,
	W = 0.000 deg,	P = 30.000 deg,	R = 138.529 deg
};
P[123]{
   GP1:
	UF : 0, UT : 1,		CONFIG : 'N U T, 0, 0, 0',
	X = 1145.784  mm,	Y = -173.421  mm,	Z = -252.534  mm,
	W = 0.000 deg,	P = 30.000 deg,	R = 143.864 deg
};
P[124]{
   GP1:
	UF : 0, UT : 1,		CONFIG : 'N U T, 0, 0, 0',
	X = 1147.767  mm,	Y = -171.417  mm,	Z = -253.118  mm,
	W = 0.000 deg,	P = 30.000 deg,	R = 155.227 deg
};
P[125]{
   GP1:
	UF : 0, UT : 1,		CONFIG : 'N U T, 0, 0, 0',
	X = 1149.806  mm,	Y = -169.415  mm,	Z = -253.706  mm,
	W = 0.000 deg,	P = 30.000 deg,	R = 166.755 deg
};
P[126]{
   GP1:
	UF : 0, UT : 1,		CONFIG : 'N U T, 0, 0, 0',
	X = 1151.836  mm,	Y = -167.349  mm,	Z = -254.276  mm,
	W = 0.000 deg,	P = 30.000 deg,	R = 178.077 deg
};
P[127]{
   GP1:
	UF : 0, UT : 1,		CONFIG : 'N U T, 0, 0, 0',
	X = 1153.596  mm,	Y = -165.267  mm,	Z = -254.752  mm,
	W = 0.000 deg,	P = 30.000 deg,	R = 178.077 deg
};
P[128]{
   GP1:
	UF : 0, UT : 1,		CONFIG : 'N U T, 0, 0, 0',
	X = 1155.258  mm,	Y = -163.171  mm,	Z = -255.198  mm,
	W = 0.000 deg,	P = 30.000 deg,	R = 178.077 deg
};
P[129]{
   GP1:
	UF : 0, UT : 1,		CONFIG : 'N U T, 0, 0, 0',
	X = 1156.665  mm,	Y = -161.009  mm,	Z = -255.554  mm,
	W = 0.000 deg,	P = 30.000 deg,	R = 178.077 deg
};
P[130]{
   GP1:
	UF : 0, UT : 1,		CONFIG : 'N U T, 0, 0, 0',
	X = 1157.796  mm,	Y = -158.826  mm,	Z = -255.828  mm,
	W = 0.000 deg,	P = 30.000 deg,	R = 178.077 deg
};
P[131]{
   GP1:
	UF : 0, UT : 1,		CONFIG : 'N U T, 0, 0, 0',
	X = 1158.657  mm,	Y = -156.612  mm,	Z = -256.022  mm,
	W = 0.000 deg,	P = 30.000 deg,	R = 178.077 deg
};
P[132]{
   GP1:
	UF : 0, UT : 1,		CONFIG : 'N U T, 0, 0, 0',
	X = 1159.225  mm,	Y = -154.375  mm,	Z = -256.144  mm,
	W = 0.000 deg,	P = 30.000 deg,	R = 178.077 deg
};
P[133]{
   GP1:
	UF : 0, UT : 1,		CONFIG : 'N U T, 0, 0, 0',
	X = 1159.504  mm,	Y = -152.218  mm,	Z = -256.190  mm,
	W = 0.000 deg,	P = 30.000 deg,	R = 178.077 deg
};
P[134]{
   GP1:
	UF : 0, UT : 1,		CONFIG : 'N U T, 0, 0, 0',
	X = 1159.694  mm,	Y = -150.137  mm,	Z = -256.215  mm,
	W = 0.000 deg,	P = 30.000 deg,	R = 178.077 deg
};
P[135]{
   GP1:
	UF : 0, UT : 1,		CONFIG : 'N U T, 0, 0, 0',
	X = 1159.789  mm,	Y = -148.075  mm,	Z = -256.220  mm,
	W = 0.000 deg,	P = 30.000 deg,	R = 178.077 deg
};
P[136]{
   GP1:
	UF : 0, UT : 1,		CONFIG : 'N U T, 0, 0, 0',
	X = 1155.851  mm,	Y = -145.951  mm,	Z = -256.223  mm,
	W = 0.000 deg,	P = 30.000 deg,	R = 178.077 deg
};
P[137]{
   GP1:
	UF : 0, UT : 1,		CONFIG : 'N U T, 0, 0, 0',
	X = 1155.889  mm,	Y = -143.971  mm,	Z = -256.223  mm,
	W = 0.000 deg,	P = 30.000 deg,	R = 178.077 deg
};
P[138]{
   GP1:
	UF : 0, UT : 1,		CONFIG : 'N U T, 0, 0, 0',
	X = 1155.909  mm,	Y = -141.981  mm,	Z = -256.220  mm,
	W = 0.000 deg,	P = 30.000 deg,	R = 178.077 deg
};
P[139]{
   GP1:
	UF : 0, UT : 1,		CONFIG : 'N U T, 0, 0, 0',
	X = 1155.927  mm,	Y = -139.986  mm,	Z = -256.216  mm,
	W = 0.000 deg,	P = 30.000 deg,	R = 178.077 deg
};
P[140]{
   GP1:
	UF : 0, UT : 1,		CONFIG : 'N U T, 0, 0, 0',
	X = 1155.936  mm,	Y = -137.995  mm,	Z = -256.207  mm,
	W = 0.000 deg,	P = 30.000 deg,	R = 178.077 deg
};
P[141]{
   GP1:
	UF : 0, UT : 1,		CONFIG : 'N U T, 0, 0, 0',
	X = 1155.937  mm,	Y = -136.000  mm,	Z = -256.186  mm,
	W = 0.000 deg,	P = 30.000 deg,	R = 178.077 deg
};
P[142]{
   GP1:
	UF : 0, UT : 1,		CONFIG : 'N U T, 0, 0, 0',
	X = 1155.937  mm,	Y = -134.000  mm,	Z = -256.159  mm,
	W = 0.000 deg,	P = 30.000 deg,	R = 178.077 deg
};
P[143]{
   GP1:
	UF : 0, UT : 1,		CONFIG : 'N U T, 0, 0, 0',
	X = 1155.936  mm,	Y = -132.001  mm,	Z = -256.127  mm,
	W = 0.000 deg,	P = 30.000 deg,	R = 178.077 deg
};
P[144]{
   GP1:
	UF : 0, UT : 1,		CONFIG : 'N U T, 0, 0, 0',
	X = 1155.934  mm,	Y = -130.004  mm,	Z = -256.092  mm,
	W = 0.000 deg,	P = 30.000 deg,	R = 178.077 deg
};
P[145]{
   GP1:
	UF : 0, UT : 1,		CONFIG : 'N U T, 0, 0, 0',
	X = 1155.927  mm,	Y = -128.013  mm,	Z = -256.054  mm,
	W = 0.000 deg,	P = 30.000 deg,	R = 178.077 deg
};
P[146]{
   GP1:
	UF : 0, UT : 1,		CONFIG : 'N U T, 0, 0, 0',
	X = 1155.908  mm,	Y = -126.020  mm,	Z = -256.013  mm,
	W = 0.000 deg,	P = 30.000 deg,	R = 178.077 deg
};
P[147]{
   GP1:
	UF : 0, UT : 1,		CONFIG : 'N U T, 0, 0, 0',
	X = 1155.888  mm,	Y = -124.029  mm,	Z = -255.972  mm,
	W = 0.000 deg,	P = 30.000 deg,	R = 178.077 deg
};
P[148]{
   GP1:
	UF : 0, UT : 1,		CONFIG : 'N U T, 0, 0, 0',
	X = 1155.851  mm,	Y = -122.049  mm,	Z = -255.932  mm,
	W = 0.000 deg,	P = 30.000 deg,	R = 178.077 deg
};
P[149]{
   GP1:
	UF : 0, UT : 1,		CONFIG : 'N U T, 0, 0, 0',
	X = 1155.791  mm,	Y = -120.064  mm,	Z = -255.887  mm,
	W = 0.000 deg,	P = 30.000 deg,	R = 178.077 deg
};
P[150]{
   GP1:
	UF : 0, UT : 1,		CONFIG : 'N U T, 0, 0, 0',
	X = 1155.723  mm,	Y = -118.077  mm,	Z = -255.841  mm,
	W = 0.000 deg,	P = 30.000 deg,	R = 178.077 deg
};
P[151]{
   GP1:
	UF : 0, UT : 1,		CONFIG : 'N U T, 0, 0, 0',
	X = 1155.638  mm,	Y = -116.096  mm,	Z = -255.797  mm,
	W = 0.000 deg,	P = 30.000 deg,	R = 178.077 deg
};
P[152]{
   GP1:
	UF : 0, UT : 1,		CONFIG : 'N U T, 0, 0, 0',
	X = 1155.533  mm,	Y = -114.120  mm,	Z = -255.744  mm,
	W = 0.000 deg,	P = 30.000 deg,	R = 178.077 deg
};
P[153]{
   GP1:
	UF : 0, UT : 1,		CONFIG : 'N U T, 0, 0, 0',
	X = 1155.402  mm,	Y = -112.155  mm,	Z = -255.686  mm,
	W = 0.000 deg,	P = 30.000 deg,	R = 178.077 deg
};
P[154]{
   GP1:
	UF : 0, UT : 1,		CONFIG : 'N U T, 0, 0, 0',
	X = 1155.226  mm,	Y = -110.174  mm,	Z = -255.613  mm,
	W = 0.000 deg,	P = 30.000 deg,	R = 178.077 deg
};
P[155]{
   GP1:
	UF : 0, UT : 1,		CONFIG : 'N U T, 0, 0, 0',
	X = 1159.037  mm,	Y = -107.794  mm,	Z = -255.549  mm,
	W = 0.000 deg,	P = 30.000 deg,	R = -173.638 deg
};
P[156]{
   GP1:
	UF : 0, UT : 1,		CONFIG : 'N U T, 0, 0, 0',
	X = 1158.782  mm,	Y = -105.712  mm,	Z = -255.462  mm,
	W = 0.000 deg,	P = 30.000 deg,	R = -164.131 deg
};
P[157]{
   GP1:
	UF : 0, UT : 1,		CONFIG : 'N U T, 0, 0, 0',
	X = 1158.418  mm,	Y = -103.563  mm,	Z = -255.346  mm,
	W = 0.000 deg,	P = 30.000 deg,	R = -154.555 deg
};
P[158]{
   GP1:
	UF : 0, UT : 1,		CONFIG : 'N U T, 0, 0, 0',
	X = 1157.823  mm,	Y = -101.427  mm,	Z = -255.158  mm,
	W = 0.000 deg,	P = 30.000 deg,	R = -144.726 deg
};
P[159]{
   GP1:
	UF : 0, UT : 1,		CONFIG : 'N U T, 0, 0, 0',
	X = 1157.120  mm,	Y = -99.241  mm,	Z = -254.954  mm,
	W = 0.000 deg,	P = 30.000 deg,	R = -134.785 deg
};
P[160]{
   GP1:
	UF : 0, UT : 1,		CONFIG : 'N U T, 0, 0, 0',
	X = 1155.997  mm,	Y = -97.001  mm,	Z = -254.634  mm,
	W = 0.000 deg,	P = 30.000 deg,	R = -134.785 deg
};
P[161]{
   GP1:
	UF : 0, UT : 1,		CONFIG : 'N U T, 0, 0, 0',
	X = 1154.612  mm,	Y = -94.868  mm,	Z = -254.226  mm,
	W = 0.000 deg,	P = 30.000 deg,	R = -134.785 deg
};
P[162]{
   GP1:
	UF : 0, UT : 1,		CONFIG : 'N U T, 0, 0, 0',
	X = 1153.096  mm,	Y = -92.771  mm,	Z = -253.773  mm,
	W = 0.000 deg,	P = 30.000 deg,	R = -134.785 deg
};
P[163]{
   GP1:
	UF : 0, UT : 1,		CONFIG : 'N U T, 0, 0, 0',
	X = 1151.317  mm,	Y = -90.643  mm,	Z = -253.245  mm,
	W = 0.000 deg,	P = 30.000 deg,	R = -134.785 deg
};
P[164]{
   GP1:
	UF : 0, UT : 1,		CONFIG : 'N U T, 0, 0, 0',
	X = 1149.248  mm,	Y = -88.595  mm,	Z = -252.596  mm,
	W = 0.000 deg,	P = 30.000 deg,	R = -134.785 deg
};
P[165]{
   GP1:
	UF : 0, UT : 1,		CONFIG : 'N U T, 0, 0, 0',
	X = 1144.508  mm,	Y = -89.438  mm,	Z = -251.981  mm,
	W = 0.000 deg,	P = 30.000 deg,	R = -134.785 deg
};
P[166]{
   GP1:
	UF : 0, UT : 1,		CONFIG : 'N U T, 0, 0, 0',
	X = 1142.350  mm,	Y = -87.489  mm,	Z = -251.271  mm,
	W = 0.000 deg,	P = 30.000 deg,	R = -134.785 deg
};
P[167]{
   GP1:
	UF : 0, UT : 1,		CONFIG : 'N U T, 0, 0, 0',
	X = 1140.097  mm,	Y = -85.483  mm,	Z = -250.529  mm,
	W = 0.000 deg,	P = 30.000 deg,	R = -134.785 deg
};
P[168]{
   GP1:
	UF : 0, UT : 1,		CONFIG : 'N U T, 0, 0, 0',
	X = 1137.936  mm,	Y = -83.495  mm,	Z = -249.794  mm,
	W = 0.000 deg,	P = 30.000 deg,	R = -134.785 deg
};
P[169]{
   GP1:
	UF : 0, UT : 1,		CONFIG : 'N U T, 0, 0, 0',
	X = 1135.665  mm,	Y = -81.544  mm,	Z = -248.992  mm,
	W = 0.000 deg,	P = 30.000 deg,	R = -134.785 deg
};
P[170]{
   GP1:
	UF : 0, UT : 1,		CONFIG : 'N U T, 0, 0, 0',
	X = 1133.136  mm,	Y = -79.543  mm,	Z = -248.198  mm,
	W = 0.000 deg,	P = 30.000 deg,	R = -134.785 deg
};
P[171]{
   GP1:
	UF : 0, UT : 1,		CONFIG : 'N U T, 0, 0, 0',
	X = 1130.803  mm,	Y = -77.533  mm,	Z = -247.497  mm,
	W = 0.000 deg,	P = 30.000 deg,	R = -139.224 deg
};
P[172]{
   GP1:
	UF : 0, UT : 1,		CONFIG : 'N U T, 0, 0, 0',
	X = 1128.327  mm,	Y = -75.516  mm,	Z = -246.795  mm,
	W = 0.000 deg,	P = 30.000 deg,	R = -153.779 deg
};
P[173]{
   GP1:
	UF : 0, UT : 1,		CONFIG : 'N U T, 0, 0, 0',
	X = 1126.026  mm,	Y = -73.417  mm,	Z = -246.205  mm,
	W = 0.000 deg,	P = 30.000 deg,	R = -167.358 deg
};
P[174]{
   GP1:
	UF : 0, UT : 1,		CONFIG : 'N U T, 0, 0, 0',
	X = 1124.093  mm,	Y = -71.295  mm,	Z = -245.765  mm,
	W = 0.000 deg,	P = 30.000 deg,	R = -179.651 deg
};
P[175]{
   GP1:
	UF : 0, UT : 1,		CONFIG : 'N U T, 0, 0, 0',
	X = 1122.411  mm,	Y = -69.162  mm,	Z = -245.422  mm,
	W = 0.000 deg,	P = 30.000 deg,	R = -179.651 deg
};
P[176]{
   GP1:
	UF : 0, UT : 1,		CONFIG : 'N U T, 0, 0, 0',
	X = 1120.980  mm,	Y = -66.911  mm,	Z = -245.187  mm,
	W = 0.000 deg,	P = 30.000 deg,	R = -179.651 deg
};
P[177]{
   GP1:
	UF : 0, UT : 1,		CONFIG : 'N U T, 0, 0, 0',
	X = 1120.090  mm,	Y = -64.621  mm,	Z = -245.049  mm,
	W = 0.000 deg,	P = 30.000 deg,	R = -179.651 deg
};
P[178]{
   GP1:
	UF : 0, UT : 1,		CONFIG : 'N U T, 0, 0, 0',
	X = 1119.493  mm,	Y = -62.392  mm,	Z = -244.976  mm,
	W = 0.000 deg,	P = 30.000 deg,	R = -179.651 deg
};
P[179]{
   GP1:
	UF : 0, UT : 1,		CONFIG : 'N U T, 0, 0, 0',
	X = 1119.201  mm,	Y = -60.198  mm,	Z = -244.944  mm,
	W = 0.000 deg,	P = 30.000 deg,	R = -179.651 deg
};
P[180]{
   GP1:
	UF : 0, UT : 1,		CONFIG : 'N U T, 0, 0, 0',
	X = 1119.059  mm,	Y = -58.102  mm,	Z = -244.921  mm,
	W = 0.000 deg,	P = 30.000 deg,	R = -179.651 deg
};
P[181]{
   GP1:
	UF : 0, UT : 1,		CONFIG : 'N U T, 0, 0, 0',
	X = 1118.987  mm,	Y = -56.056  mm,	Z = -244.908  mm,
	W = 0.000 deg,	P = 30.000 deg,	R = -179.651 deg
};
P[182]{
   GP1:
	UF : 0, UT : 1,		CONFIG : 'N U T, 0, 0, 0',
	X = 1118.944  mm,	Y = -54.038  mm,	Z = -244.896  mm,
	W = 0.000 deg,	P = 30.000 deg,	R = -179.651 deg
};
P[183]{
   GP1:
	UF : 0, UT : 1,		CONFIG : 'N U T, 0, 0, 0',
	X = 1118.910  mm,	Y = -52.027  mm,	Z = -244.886  mm,
	W = 0.000 deg,	P = 30.000 deg,	R = -179.651 deg
};
P[184]{
   GP1:
	UF : 0, UT : 1,		CONFIG : 'N U T, 0, 0, 0',
	X = 1122.890  mm,	Y = -49.989  mm,	Z = -244.880  mm,
	W = 0.000 deg,	P = 30.000 deg,	R = -179.651 deg
};
P[185]{
   GP1:
	UF : 0, UT : 1,		CONFIG : 'N U T, 0, 0, 0',
	X = 1122.889  mm,	Y = -48.001  mm,	Z = -244.868  mm,
	W = 0.000 deg,	P = 30.000 deg,	R = -179.651 deg
};
P[186]{
   GP1:
	UF : 0, UT : 1,		CONFIG : 'N U T, 0, 0, 0',
	X = 1122.891  mm,	Y = -46.004  mm,	Z = -244.859  mm,
	W = 0.000 deg,	P = 30.000 deg,	R = -179.651 deg
};
P[187]{
   GP1:
	UF : 0, UT : 1,		CONFIG : 'N U T, 0, 0, 0',
	X = 1122.897  mm,	Y = -44.012  mm,	Z = -244.850  mm,
	W = 0.000 deg,	P = 30.000 deg,	R = -179.651 deg
};
P[188]{
   GP1:
	UF : 0, UT : 1,		CONFIG : 'N U T, 0, 0, 0',
	X = 1122.914  mm,	Y = -42.019  mm,	Z = -244.840  mm,
	W = 0.000 deg,	P = 30.000 deg,	R = -179.651 deg
};
P[189]{
   GP1:
	UF : 0, UT : 1,		CONFIG : 'N U T, 0, 0, 0',
	X = 1122.935  mm,	Y = -40.022  mm,	Z = -244.829  mm,
	W = 0.000 deg,	P = 30.000 deg,	R = -179.651 deg
};
P[190]{
   GP1:
	UF : 0, UT : 1,		CONFIG : 'N U T, 0, 0, 0',
	X = 1122.958  mm,	Y = -38.024  mm,	Z = -244.815  mm,
	W = 0.000 deg,	P = 30.000 deg,	R = -179.651 deg
};
P[191]{
   GP1:
	UF : 0, UT : 1,		CONFIG : 'N U T, 0, 0, 0',
	X = 1122.984  mm,	Y = -36.029  mm,	Z = -244.795  mm,
	W = 0.000 deg,	P = 30.000 deg,	R = -179.651 deg
};
P[192]{
   GP1:
	UF : 0, UT : 1,		CONFIG : 'N U T, 0, 0, 0',
	X = 1123.016  mm,	Y = -34.039  mm,	Z = -244.775  mm,
	W = 0.000 deg,	P = 30.000 deg,	R = -179.651 deg
};
P[193]{
   GP1:
	UF : 0, UT : 1,		CONFIG : 'N U T, 0, 0, 0',
	X = 1123.060  mm,	Y = -32.050  mm,	Z = -244.754  mm,
	W = 0.000 deg,	P = 30.000 deg,	R = -179.651 deg
};
P[194]{
   GP1:
	UF : 0, UT : 1,		CONFIG : 'N U T, 0, 0, 0',
	X = 1123.115  mm,	Y = -30.055  mm,	Z = -244.734  mm,
	W = 0.000 deg,	P = 30.000 deg,	R = -179.651 deg
};
P[195]{
   GP1:
	UF : 0, UT : 1,		CONFIG : 'N U T, 0, 0, 0',
	X = 1123.170  mm,	Y = -28.063  mm,	Z = -244.713  mm,
	W = 0.000 deg,	P = 30.000 deg,	R = -179.651 deg
};
P[196]{
   GP1:
	UF : 0, UT : 1,		CONFIG : 'N U T, 0, 0, 0',
	X = 1123.240  mm,	Y = -26.086  mm,	Z = -244.697  mm,
	W = 0.000 deg,	P = 30.000 deg,	R = -179.651 deg
};
P[197]{
   GP1:
	UF : 0, UT : 1,		CONFIG : 'N U T, 0, 0, 0',
	X = 1123.341  mm,	Y = -24.106  mm,	Z = -244.682  mm,
	W = 0.000 deg,	P = 30.000 deg,	R = -179.651 deg
};
P[198]{
   GP1:
	UF : 0, UT : 1,		CONFIG : 'N U T, 0, 0, 0',
	X = 1123.451  mm,	Y = -22.117  mm,	Z = -244.669  mm,
	W = 0.000 deg,	P = 30.000 deg,	R = -179.651 deg
};
P[199]{
   GP1:
	UF : 0, UT : 1,		CONFIG : 'N U T, 0, 0, 0',
	X = 1123.573  mm,	Y = -20.127  mm,	Z = -244.657  mm,
	W = 0.000 deg,	P = 30.000 deg,	R = -179.651 deg
};
P[200]{
   GP1:
	UF : 0, UT : 1,		CONFIG : 'N U T, 0, 0, 0',
	X = 1119.715  mm,	Y = -17.839  mm,	Z = -244.643  mm,
	W = 0.000 deg,	P = 30.000 deg,	R = 172.400 deg
};
P[201]{
   GP1:
	UF : 0, UT : 1,		CONFIG : 'N U T, 0, 0, 0',
	X = 1119.911  mm,	Y = -15.777  mm,	Z = -244.635  mm,
	W = 0.000 deg,	P = 30.000 deg,	R = 163.955 deg
};
P[202]{
   GP1:
	UF : 0, UT : 1,		CONFIG : 'N U T, 0, 0, 0',
	X = 1120.178  mm,	Y = -13.709  mm,	Z = -244.638  mm,
	W = 0.000 deg,	P = 30.000 deg,	R = 155.478 deg
};
P[203]{
   GP1:
	UF : 0, UT : 1,		CONFIG : 'N U T, 0, 0, 0',
	X = 1120.526  mm,	Y = -11.605  mm,	Z = -244.644  mm,
	W = 0.000 deg,	P = 30.000 deg,	R = 146.958 deg
};
P[204]{
   GP1:
	UF : 0, UT : 1,		CONFIG : 'N U T, 0, 0, 0',
	X = 1121.045  mm,	Y = -9.431  mm,	Z = -244.688  mm,
	W = 0.000 deg,	P = 30.000 deg,	R = 138.314 deg
};
P[205]{
   GP1:
	UF : 0, UT : 1,		CONFIG : 'N U T, 0, 0, 0',
	X = 1121.817  mm,	Y = -7.257  mm,	Z = -244.804  mm,
	W = 0.000 deg,	P = 30.000 deg,	R = 138.314 deg
};
P[206]{
   GP1:
	UF : 0, UT : 1,		CONFIG : 'N U T, 0, 0, 0',
	X = 1122.765  mm,	Y = -5.123  mm,	Z = -244.970  mm,
	W = 0.000 deg,	P = 30.000 deg,	R = 138.314 deg
};
P[207]{
   GP1:
	UF : 0, UT : 1,		CONFIG : 'N U T, 0, 0, 0',
	X = 1123.899  mm,	Y = -2.991  mm,	Z = -245.179  mm,
	W = 0.000 deg,	P = 30.000 deg,	R = 138.314 deg
};
P[208]{
   GP1:
	UF : 0, UT : 1,		CONFIG : 'N U T, 0, 0, 0',
	X = 1125.252  mm,	Y = -0.866  mm,	Z = -245.409  mm,
	W = 0.000 deg,	P = 30.000 deg,	R = 138.314 deg
};
P[209]{
   GP1:
	UF : 0, UT : 1,		CONFIG : 'N U T, 0, 0, 0',
	X = 1126.799  mm,	Y = 1.224  mm,	Z = -245.726  mm,
	W = 0.000 deg,	P = 30.000 deg,	R = 138.314 deg
};
P[210]{
   GP1:
	UF : 0, UT : 1,		CONFIG : 'N U T, 0, 0, 0',
	X = 1128.463  mm,	Y = 3.284  mm,	Z = -246.110  mm,
	W = 0.000 deg,	P = 30.000 deg,	R = 138.314 deg
};
P[211]{
   GP1:
	UF : 0, UT : 1,		CONFIG : 'N U T, 0, 0, 0',
	X = 1130.231  mm,	Y = 5.325  mm,	Z = -246.567  mm,
	W = 0.000 deg,	P = 30.000 deg,	R = 138.314 deg
};
P[212]{
   GP1:
	UF : 0, UT : 1,		CONFIG : 'N U T, 0, 0, 0',
	X = 1134.981  mm,	Y = 4.619  mm,	Z = -247.066  mm,
	W = 0.000 deg,	P = 30.000 deg,	R = 138.314 deg
};
P[213]{
   GP1:
	UF : 0, UT : 1,		CONFIG : 'N U T, 0, 0, 0',
	X = 1136.946  mm,	Y = 6.568  mm,	Z = -247.636  mm,
	W = 0.000 deg,	P = 30.000 deg,	R = 138.314 deg
};
P[214]{
   GP1:
	UF : 0, UT : 1,		CONFIG : 'N U T, 0, 0, 0',
	X = 1139.020  mm,	Y = 8.556  mm,	Z = -248.250  mm,
	W = 0.000 deg,	P = 30.000 deg,	R = 138.314 deg
};
P[215]{
   GP1:
	UF : 0, UT : 1,		CONFIG : 'N U T, 0, 0, 0',
	X = 1141.106  mm,	Y = 10.552  mm,	Z = -248.933  mm,
	W = 0.000 deg,	P = 30.000 deg,	R = 138.314 deg
};
P[216]{
   GP1:
	UF : 0, UT : 1,		CONFIG : 'N U T, 0, 0, 0',
	X = 1143.207  mm,	Y = 12.542  mm,	Z = -249.615  mm,
	W = 0.000 deg,	P = 30.000 deg,	R = 138.314 deg
};
P[217]{
   GP1:
	UF : 0, UT : 1,		CONFIG : 'N U T, 0, 0, 0',
	X = 1145.357  mm,	Y = 14.544  mm,	Z = -250.303  mm,
	W = 0.000 deg,	P = 30.000 deg,	R = 142.589 deg
};
P[218]{
   GP1:
	UF : 0, UT : 1,		CONFIG : 'N U T, 0, 0, 0',
	X = 1147.458  mm,	Y = 16.545  mm,	Z = -250.953  mm,
	W = 0.000 deg,	P = 30.000 deg,	R = 153.881 deg
};
P[219]{
   GP1:
	UF : 0, UT : 1,		CONFIG : 'N U T, 0, 0, 0',
	X = 1149.617  mm,	Y = 18.559  mm,	Z = -251.599  mm,
	W = 0.000 deg,	P = 30.000 deg,	R = 165.285 deg
};
P[220]{
   GP1:
	UF : 0, UT : 1,		CONFIG : 'N U T, 0, 0, 0',
	X = 1151.666  mm,	Y = 20.596  mm,	Z = -252.204  mm,
	W = 0.000 deg,	P = 30.000 deg,	R = 176.305 deg
};
P[221]{
   GP1:
	UF : 0, UT : 1,		CONFIG : 'N U T, 0, 0, 0',
	X = 1153.640  mm,	Y = 22.643  mm,	Z = -252.780  mm,
	W = 0.000 deg,	P = 30.000 deg,	R = 176.305 deg
};
P[222]{
   GP1:
	UF : 0, UT : 1,		CONFIG : 'N U T, 0, 0, 0',
	X = 1155.482  mm,	Y = 24.734  mm,	Z = -253.296  mm,
	W = 0.000 deg,	P = 30.000 deg,	R = 176.305 deg
};
P[223]{
   GP1:
	UF : 0, UT : 1,		CONFIG : 'N U T, 0, 0, 0',
	X = 1157.087  mm,	Y = 26.860  mm,	Z = -253.727  mm,
	W = 0.000 deg,	P = 30.000 deg,	R = 176.305 deg
};
P[224]{
   GP1:
	UF : 0, UT : 1,		CONFIG : 'N U T, 0, 0, 0',
	X = 1158.444  mm,	Y = 29.007  mm,	Z = -254.082  mm,
	W = 0.000 deg,	P = 30.000 deg,	R = 176.305 deg
};
P[225]{
   GP1:
	UF : 0, UT : 1,		CONFIG : 'N U T, 0, 0, 0',
	X = 1159.576  mm,	Y = 31.223  mm,	Z = -254.367  mm,
	W = 0.000 deg,	P = 30.000 deg,	R = 176.305 deg
};
P[226]{
   GP1:
	UF : 0, UT : 1,		CONFIG : 'N U T, 0, 0, 0',
	X = 1160.329  mm,	Y = 33.491  mm,	Z = -254.550  mm,
	W = 0.000 deg,	P = 30.000 deg,	R = 176.305 deg
};
P[227]{
   GP1:
	UF : 0, UT : 1,		CONFIG : 'N U T, 0, 0, 0',
	X = 1160.763  mm,	Y = 35.704  mm,	Z = -254.654  mm,
	W = 0.000 deg,	P = 30.000 deg,	R = 176.305 deg
};
P[228]{
   GP1:
	UF : 0, UT : 1,		CONFIG : 'N U T, 0, 0, 0',
	X = 1160.987  mm,	Y = 37.845  mm,	Z = -254.705  mm,
	W = 0.000 deg,	P = 30.000 deg,	R = 176.305 deg
};
P[229]{
   GP1:
	UF : 0, UT : 1,		CONFIG : 'N U T, 0, 0, 0',
	X = 1157.097  mm,	Y = 40.078  mm,	Z = -254.718  mm,
	W = 0.000 deg,	P = 30.000 deg,	R = 176.305 deg
};
P[230]{
   GP1:
	UF : 0, UT : 1,		CONFIG : 'N U T, 0, 0, 0',
	X = 1157.149  mm,	Y = 42.046  mm,	Z = -254.718  mm,
	W = 0.000 deg,	P = 30.000 deg,	R = 176.305 deg
};
P[231]{
   GP1:
	UF : 0, UT : 1,		CONFIG : 'N U T, 0, 0, 0',
	X = 1157.187  mm,	Y = 44.034  mm,	Z = -254.711  mm,
	W = 0.000 deg,	P = 30.000 deg,	R = 176.305 deg
};
P[232]{
   GP1:
	UF : 0, UT : 1,		CONFIG : 'N U T, 0, 0, 0',
	X = 1157.217  mm,	Y = 46.029  mm,	Z = -254.700  mm,
	W = 0.000 deg,	P = 30.000 deg,	R = 176.305 deg
};
P[233]{
   GP1:
	UF : 0, UT : 1,		CONFIG : 'N U T, 0, 0, 0',
	X = 1157.244  mm,	Y = 48.026  mm,	Z = -254.685  mm,
	W = 0.000 deg,	P = 30.000 deg,	R = 176.305 deg
};
P[234]{
   GP1:
	UF : 0, UT : 1,		CONFIG : 'N U T, 0, 0, 0',
	X = 1157.268  mm,	Y = 50.021  mm,	Z = -254.668  mm,
	W = 0.000 deg,	P = 30.000 deg,	R = 176.305 deg
};
P[235]{
   GP1:
	UF : 0, UT : 1,		CONFIG : 'N U T, 0, 0, 0',
	X = 1157.286  mm,	Y = 52.011  mm,	Z = -254.648  mm,
	W = 0.000 deg,	P = 30.000 deg,	R = 176.305 deg
};
P[236]{
   GP1:
	UF : 0, UT : 1,		CONFIG : 'N U T, 0, 0, 0',
	X = 1157.291  mm,	Y = 54.001  mm,	Z = -254.625  mm,
	W = 0.000 deg,	P = 30.000 deg,	R = 176.305 deg
};
P[237]{
   GP1:
	UF : 0, UT : 1,		CONFIG : 'N U T, 0, 0, 0',
	X = 1157.288  mm,	Y = 55.995  mm,	Z = -254.602  mm,
	W = 0.000 deg,	P = 30.000 deg,	R = 176.305 deg
};
P[238]{
   GP1:
	UF : 0, UT : 1,		CONFIG : 'N U T, 0, 0, 0',
	X = 1157.281  mm,	Y = 57.989  mm,	Z = -254.576  mm,
	W = 0.000 deg,	P = 30.000 deg,	R = 176.305 deg
};
P[239]{
   GP1:
	UF : 0, UT : 1,		CONFIG : 'N U T, 0, 0, 0',
	X = 1157.266  mm,	Y = 59.984  mm,	Z = -254.548  mm,
	W = 0.000 deg,	P = 30.000 deg,	R = 176.305 deg
};
P[240]{
   GP1:
	UF : 0, UT : 1,		CONFIG : 'N U T, 0, 0, 0',
	X = 1157.249  mm,	Y = 61.977  mm,	Z = -254.520  mm,
	W = 0.000 deg,	P = 30.000 deg,	R = 176.305 deg
};
P[241]{
   GP1:
	UF : 0, UT : 1,		CONFIG : 'N U T, 0, 0, 0',
	X = 1157.220  mm,	Y = 63.970  mm,	Z = -254.484  mm,
	W = 0.000 deg,	P = 30.000 deg,	R = 176.305 deg
};
P[242]{
   GP1:
	UF : 0, UT : 1,		CONFIG : 'N U T, 0, 0, 0',
	X = 1157.189  mm,	Y = 65.964  mm,	Z = -254.450  mm,
	W = 0.000 deg,	P = 30.000 deg,	R = 176.305 deg
};
P[243]{
   GP1:
	UF : 0, UT : 1,		CONFIG : 'N U T, 0, 0, 0',
	X = 1157.149  mm,	Y = 67.952  mm,	Z = -254.415  mm,
	W = 0.000 deg,	P = 30.000 deg,	R = 176.305 deg
};
P[244]{
   GP1:
	UF : 0, UT : 1,		CONFIG : 'N U T, 0, 0, 0',
	X = 1157.093  mm,	Y = 69.938  mm,	Z = -254.381  mm,
	W = 0.000 deg,	P = 30.000 deg,	R = 176.305 deg
};
P[245]{
   GP1:
	UF : 0, UT : 1,		CONFIG : 'N U T, 0, 0, 0',
	X = 1157.026  mm,	Y = 71.930  mm,	Z = -254.339  mm,
	W = 0.000 deg,	P = 30.000 deg,	R = 176.305 deg
};
P[246]{
   GP1:
	UF : 0, UT : 1,		CONFIG : 'N U T, 0, 0, 0',
	X = 1156.953  mm,	Y = 73.923  mm,	Z = -254.298  mm,
	W = 0.000 deg,	P = 30.000 deg,	R = 176.305 deg
};
P[247]{
   GP1:
	UF : 0, UT : 1,		CONFIG : 'N U T, 0, 0, 0',
	X = 1156.873  mm,	Y = 75.921  mm,	Z = -254.253  mm,
	W = 0.000 deg,	P = 30.000 deg,	R = 176.305 deg
};
P[248]{
   GP1:
	UF : 0, UT : 1,		CONFIG : 'N U T, 0, 0, 0',
	X = 1156.795  mm,	Y = 77.911  mm,	Z = -254.212  mm,
	W = 0.000 deg,	P = 30.000 deg,	R = 176.305 deg
};
P[249]{
   GP1:
	UF : 0, UT : 1,		CONFIG : 'N U T, 0, 0, 0',
	X = 1160.688  mm,	Y = 80.143  mm,	Z = -254.161  mm,
	W = 0.000 deg,	P = 30.000 deg,	R = -175.038 deg
};
P[250]{
   GP1:
	UF : 0, UT : 1,		CONFIG : 'N U T, 0, 0, 0',
	X = 1160.496  mm,	Y = 82.201  mm,	Z = -254.086  mm,
	W = 0.000 deg,	P = 30.000 deg,	R = -165.537 deg
};
P[251]{
   GP1:
	UF : 0, UT : 1,		CONFIG : 'N U T, 0, 0, 0',
	X = 1160.266  mm,	Y = 84.295  mm,	Z = -253.992  mm,
	W = 0.000 deg,	P = 30.000 deg,	R = -156.018 deg
};
P[252]{
   GP1:
	UF : 0, UT : 1,		CONFIG : 'N U T, 0, 0, 0',
	X = 1159.850  mm,	Y = 86.485  mm,	Z = -253.862  mm,
	W = 0.000 deg,	P = 30.000 deg,	R = -146.379 deg
};
P[253]{
   GP1:
	UF : 0, UT : 1,		CONFIG : 'N U T, 0, 0, 0',
	X = 1159.165  mm,	Y = 88.693  mm,	Z = -253.655  mm,
	W = 0.000 deg,	P = 30.000 deg,	R = -136.433 deg
};
P[254]{
   GP1:
	UF : 0, UT : 1,		CONFIG : 'N U T, 0, 0, 0',
	X = 1158.212  mm,	Y = 90.914  mm,	Z = -253.373  mm,
	W = 0.000 deg,	P = 30.000 deg,	R = -136.433 deg
};
P[255]{
   GP1:
	UF : 0, UT : 1,		CONFIG : 'N U T, 0, 0, 0',
	X = 1156.881  mm,	Y = 93.134  mm,	Z = -252.983  mm,
	W = 0.000 deg,	P = 30.000 deg,	R = -136.433 deg
};
P[256]{
   GP1:
	UF : 0, UT : 1,		CONFIG : 'N U T, 0, 0, 0',
	X = 1155.237  mm,	Y = 95.253  mm,	Z = -252.485  mm,
	W = 0.000 deg,	P = 30.000 deg,	R = -136.433 deg
};
P[257]{
   GP1:
	UF : 0, UT : 1,		CONFIG : 'N U T, 0, 0, 0',
	X = 1153.481  mm,	Y = 97.365  mm,	Z = -251.939  mm,
	W = 0.000 deg,	P = 30.000 deg,	R = -136.433 deg
};
P[258]{
   GP1:
	UF : 0, UT : 1,		CONFIG : 'N U T, 0, 0, 0',
	X = 1148.538  mm,	Y = 96.574  mm,	Z = -251.258  mm,
	W = 0.000 deg,	P = 30.000 deg,	R = -136.433 deg
};
P[259]{
   GP1:
	UF : 0, UT : 1,		CONFIG : 'N U T, 0, 0, 0',
	X = 1146.585  mm,	Y = 98.541  mm,	Z = -250.601  mm,
	W = 0.000 deg,	P = 30.000 deg,	R = -136.433 deg
};
P[260]{
   GP1:
	UF : 0, UT : 1,		CONFIG : 'N U T, 0, 0, 0',
	X = 1144.329  mm,	Y = 100.521  mm,	Z = -249.838  mm,
	W = 0.000 deg,	P = 30.000 deg,	R = -136.433 deg
};
P[261]{
   GP1:
	UF : 0, UT : 1,		CONFIG : 'N U T, 0, 0, 0',
	X = 1142.185  mm,	Y = 102.549  mm,	Z = -249.126  mm,
	W = 0.000 deg,	P = 30.000 deg,	R = -136.433 deg
};
P[262]{
   GP1:
	UF : 0, UT : 1,		CONFIG : 'N U T, 0, 0, 0',
	X = 1140.081  mm,	Y = 104.550  mm,	Z = -248.399  mm,
	W = 0.000 deg,	P = 30.000 deg,	R = -136.433 deg
};
P[263]{
   GP1:
	UF : 0, UT : 1,		CONFIG : 'N U T, 0, 0, 0',
	X = 1138.034  mm,	Y = 106.494  mm,	Z = -247.649  mm,
	W = 0.000 deg,	P = 30.000 deg,	R = -136.433 deg
};
P[264]{
   GP1:
	UF : 0, UT : 1,		CONFIG : 'N U T, 0, 0, 0',
	X = 1135.572  mm,	Y = 108.487  mm,	Z = -246.870  mm,
	W = 0.000 deg,	P = 30.000 deg,	R = -136.433 deg
};
P[265]{
   GP1:
	UF : 0, UT : 1,		CONFIG : 'N U T, 0, 0, 0',
	X = 1133.414  mm,	Y = 110.487  mm,	Z = -246.212  mm,
	W = 0.000 deg,	P = 30.000 deg,	R = -136.433 deg
};
P[266]{
   GP1:
	UF : 0, UT : 1,		CONFIG : 'N U T, 0, 0, 0',
	X = 1130.927  mm,	Y = 112.502  mm,	Z = -245.509  mm,
	W = 0.000 deg,	P = 30.000 deg,	R = -136.433 deg
};
P[267]{
   GP1:
	UF : 0, UT : 1,		CONFIG : 'N U T, 0, 0, 0',
	X = 1128.810  mm,	Y = 114.563  mm,	Z = -244.974  mm,
	W = 0.000 deg,	P = 30.000 deg,	R = -145.121 deg
};
P[268]{
   GP1:
	UF : 0, UT : 1,		CONFIG : 'N U T, 0, 0, 0',
	X = 1126.679  mm,	Y = 116.612  mm,	Z = -244.453  mm,
	W = 0.000 deg,	P = 30.000 deg,	R = -158.490 deg
};
P[269]{
   GP1:
	UF : 0, UT : 1,		CONFIG : 'N U T, 0, 0, 0',
	X = 1124.777  mm,	Y = 118.757  mm,	Z = -244.052  mm,
	W = 0.000 deg,	P = 30.000 deg,	R = -170.811 deg
};
P[270]{
   GP1:
	UF : 0, UT : 1,		CONFIG : 'N U T, 0, 0, 0',
	X = 1123.200  mm,	Y = 121.019  mm,	Z = -243.791  mm,
	W = 0.000 deg,	P = 30.000 deg,	R = 178.001 deg
};
P[271]{
   GP1:
	UF : 0, UT : 1,		CONFIG : 'N U T, 0, 0, 0',
	X = 1122.230  mm,	Y = 123.274  mm,	Z = -243.629  mm,
	W = 0.000 deg,	P = 30.000 deg,	R = 178.001 deg
};
P[272]{
   GP1:
	UF : 0, UT : 1,		CONFIG : 'N U T, 0, 0, 0',
	X = 1121.448  mm,	Y = 125.503  mm,	Z = -243.495  mm,
	W = 0.000 deg,	P = 30.000 deg,	R = 178.001 deg
};
P[273]{
   GP1:
	UF : 0, UT : 1,		CONFIG : 'N U T, 0, 0, 0',
	X = 1121.083  mm,	Y = 127.745  mm,	Z = -243.432  mm,
	W = 0.000 deg,	P = 30.000 deg,	R = 178.001 deg
};
P[274]{
   GP1:
	UF : 0, UT : 1,		CONFIG : 'N U T, 0, 0, 0',
	X = 1120.876  mm,	Y = 129.861  mm,	Z = -243.386  mm,
	W = 0.000 deg,	P = 30.000 deg,	R = 178.001 deg
};
P[275]{
   GP1:
	UF : 0, UT : 1,		CONFIG : 'N U T, 0, 0, 0',
	X = 1120.790  mm,	Y = 131.932  mm,	Z = -243.351  mm,
	W = 0.000 deg,	P = 30.000 deg,	R = 178.001 deg
};
P[276]{
   GP1:
	UF : 0, UT : 1,		CONFIG : 'N U T, 0, 0, 0',
	X = 1120.735  mm,	Y = 133.952  mm,	Z = -243.315  mm,
	W = 0.000 deg,	P = 30.000 deg,	R = 178.001 deg
};
P[277]{
   GP1:
	UF : 0, UT : 1,		CONFIG : 'N U T, 0, 0, 0',
	X = 1120.693  mm,	Y = 135.964  mm,	Z = -243.282  mm,
	W = 0.000 deg,	P = 30.000 deg,	R = 178.001 deg
};
P[278]{
   GP1:
	UF : 0, UT : 1,		CONFIG : 'N U T, 0, 0, 0',
	X = 1120.664  mm,	Y = 137.978  mm,	Z = -243.252  mm,
	W = 0.000 deg,	P = 30.000 deg,	R = 178.001 deg
};
P[279]{
   GP1:
	UF : 0, UT : 1,		CONFIG : 'N U T, 0, 0, 0',
	X = 1120.649  mm,	Y = 139.987  mm,	Z = -243.226  mm,
	W = 0.000 deg,	P = 30.000 deg,	R = 178.001 deg
};
P[280]{
   GP1:
	UF : 0, UT : 1,		CONFIG : 'N U T, 0, 0, 0',
	X = 1120.637  mm,	Y = 141.992  mm,	Z = -243.195  mm,
	W = 0.000 deg,	P = 30.000 deg,	R = 178.001 deg
};
P[281]{
   GP1:
	UF : 0, UT : 1,		CONFIG : 'N U T, 0, 0, 0',
	X = 1120.632  mm,	Y = 143.999  mm,	Z = -243.163  mm,
	W = 0.000 deg,	P = 30.000 deg,	R = 178.001 deg
};
P[282]{
   GP1:
	UF : 0, UT : 1,		CONFIG : 'N U T, 0, 0, 0',
	X = 1120.636  mm,	Y = 146.011  mm,	Z = -243.130  mm,
	W = 0.000 deg,	P = 30.000 deg,	R = 178.001 deg
};
P[283]{
   GP1:
	UF : 0, UT : 1,		CONFIG : 'N U T, 0, 0, 0',
	X = 1120.654  mm,	Y = 148.031  mm,	Z = -243.103  mm,
	W = 0.000 deg,	P = 30.000 deg,	R = 178.001 deg
};
P[284]{
   GP1:
	UF : 0, UT : 1,		CONFIG : 'N U T, 0, 0, 0',
	X = 1120.699  mm,	Y = 150.046  mm,	Z = -243.073  mm,
	W = 0.000 deg,	P = 30.000 deg,	R = 178.001 deg
};
P[285]{
   GP1:
	UF : 0, UT : 1,		CONFIG : 'N U T, 0, 0, 0',
	X = 1120.746  mm,	Y = 152.050  mm,	Z = -243.048  mm,
	W = 0.000 deg,	P = 30.000 deg,	R = 178.001 deg
};
P[286]{
   GP1:
	UF : 0, UT : 1,		CONFIG : 'N U T, 0, 0, 0',
	X = 1120.799  mm,	Y = 154.058  mm,	Z = -243.028  mm,
	W = 0.000 deg,	P = 30.000 deg,	R = 178.001 deg
};
P[287]{
   GP1:
	UF : 0, UT : 1,		CONFIG : 'N U T, 0, 0, 0',
	X = 1124.860  mm,	Y = 155.930  mm,	Z = -243.015  mm,
	W = 0.000 deg,	P = 30.000 deg,	R = 178.001 deg
};
P[288]{
   GP1:
	UF : 0, UT : 1,		CONFIG : 'N U T, 0, 0, 0',
	X = 1124.936  mm,	Y = 157.916  mm,	Z = -243.008  mm,
	W = 0.000 deg,	P = 30.000 deg,	R = 178.001 deg
};
P[289]{
   GP1:
	UF : 0, UT : 1,		CONFIG : 'N U T, 0, 0, 0',
	X = 1125.026  mm,	Y = 159.906  mm,	Z = -243.008  mm,
	W = 0.000 deg,	P = 30.000 deg,	R = 178.001 deg
};
P[290]{
   GP1:
	UF : 0, UT : 1,		CONFIG : 'N U T, 0, 0, 0',
	X = 1125.124  mm,	Y = 161.911  mm,	Z = -243.011  mm,
	W = 0.000 deg,	P = 30.000 deg,	R = 178.001 deg
};
P[291]{
   GP1:
	UF : 0, UT : 1,		CONFIG : 'N U T, 0, 0, 0',
	X = 1125.205  mm,	Y = 163.906  mm,	Z = -243.018  mm,
	W = 0.000 deg,	P = 30.000 deg,	R = 178.001 deg
};
P[292]{
   GP1:
	UF : 0, UT : 1,		CONFIG : 'N U T, 0, 0, 0',
	X = 1125.311  mm,	Y = 165.881  mm,	Z = -243.025  mm,
	W = 0.000 deg,	P = 30.000 deg,	R = 178.001 deg
};
P[293]{
   GP1:
	UF : 0, UT : 1,		CONFIG : 'N U T, 0, 0, 0',
	X = 1125.440  mm,	Y = 167.858  mm,	Z = -243.035  mm,
	W = 0.000 deg,	P = 30.000 deg,	R = 178.001 deg
};
P[294]{
   GP1:
	UF : 0, UT : 1,		CONFIG : 'N U T, 0, 0, 0',
	X = 1125.593  mm,	Y = 169.842  mm,	Z = -243.042  mm,
	W = 0.000 deg,	P = 30.000 deg,	R = 178.001 deg
};
P[295]{
   GP1:
	UF : 0, UT : 1,		CONFIG : 'N U T, 0, 0, 0',
	X = 1121.770  mm,	Y = 172.178  mm,	Z = -243.053  mm,
	W = 0.000 deg,	P = 30.000 deg,	R = 170.470 deg
};
P[296]{
   GP1:
	UF : 0, UT : 1,		CONFIG : 'N U T, 0, 0, 0',
	X = 1121.972  mm,	Y = 174.245  mm,	Z = -243.064  mm,
	W = 0.000 deg,	P = 30.000 deg,	R = 162.180 deg
};
P[297]{
   GP1:
	UF : 0, UT : 1,		CONFIG : 'N U T, 0, 0, 0',
	X = 1122.291  mm,	Y = 176.375  mm,	Z = -243.077  mm,
	W = 0.000 deg,	P = 30.000 deg,	R = 153.837 deg
};
P[298]{
   GP1:
	UF : 0, UT : 1,		CONFIG : 'N U T, 0, 0, 0',
	X = 1122.787  mm,	Y = 178.515  mm,	Z = -243.099  mm,
	W = 0.000 deg,	P = 30.000 deg,	R = 145.366 deg
};
P[299]{
   GP1:
	UF : 0, UT : 1,		CONFIG : 'N U T, 0, 0, 0',
	X = 1123.433  mm,	Y = 180.660  mm,	Z = -243.163  mm,
	W = 0.000 deg,	P = 30.000 deg,	R = 136.745 deg
};
P[300]{
   GP1:
	UF : 0, UT : 1,		CONFIG : 'N U T, 0, 0, 0',
	X = 1124.294  mm,	Y = 182.822  mm,	Z = -243.288  mm,
	W = 0.000 deg,	P = 30.000 deg,	R = 136.745 deg
};
P[301]{
   GP1:
	UF : 0, UT : 1,		CONFIG : 'N U T, 0, 0, 0',
	X = 1125.378  mm,	Y = 184.976  mm,	Z = -243.466  mm,
	W = 0.000 deg,	P = 30.000 deg,	R = 136.745 deg
};
P[302]{
   GP1:
	UF : 0, UT : 1,		CONFIG : 'N U T, 0, 0, 0',
	X = 1126.700  mm,	Y = 187.126  mm,	Z = -243.698  mm,
	W = 0.000 deg,	P = 30.000 deg,	R = 136.745 deg
};
P[303]{
   GP1:
	UF : 0, UT : 1,		CONFIG : 'N U T, 0, 0, 0',
	X = 1128.263  mm,	Y = 189.218  mm,	Z = -243.968  mm,
	W = 0.000 deg,	P = 30.000 deg,	R = 136.745 deg
};
P[304]{
   GP1:
	UF : 0, UT : 1,		CONFIG : 'N U T, 0, 0, 0',
	X = 1129.872  mm,	Y = 191.264  mm,	Z = -244.292  mm,
	W = 0.000 deg,	P = 30.000 deg,	R = 136.745 deg
};
P[305]{
   GP1:
	UF : 0, UT : 1,		CONFIG : 'N U T, 0, 0, 0',
	X = 1131.628  mm,	Y = 193.340  mm,	Z = -244.708  mm,
	W = 0.000 deg,	P = 30.000 deg,	R = 136.745 deg
};
P[306]{
   GP1:
	UF : 0, UT : 1,		CONFIG : 'N U T, 0, 0, 0',
	X = 1136.459  mm,	Y = 192.600  mm,	Z = -245.227  mm,
	W = 0.000 deg,	P = 30.000 deg,	R = 136.745 deg
};
P[307]{
   GP1:
	UF : 0, UT : 1,		CONFIG : 'N U T, 0, 0, 0',
	X = 1138.441  mm,	Y = 194.579  mm,	Z = -245.786  mm,
	W = 0.000 deg,	P = 30.000 deg,	R = 136.745 deg
};
P[308]{
   GP1:
	UF : 0, UT : 1,		CONFIG : 'N U T, 0, 0, 0',
	X = 1140.444  mm,	Y = 196.546  mm,	Z = -246.379  mm,
	W = 0.000 deg,	P = 30.000 deg,	R = 136.745 deg
};
P[309]{
   GP1:
	UF : 0, UT : 1,		CONFIG : 'N U T, 0, 0, 0',
	X = 1142.614  mm,	Y = 198.521  mm,	Z = -247.048  mm,
	W = 0.000 deg,	P = 30.000 deg,	R = 136.745 deg
};
P[310]{
   GP1:
	UF : 0, UT : 1,		CONFIG : 'N U T, 0, 0, 0',
	X = 1144.793  mm,	Y = 200.503  mm,	Z = -247.775  mm,
	W = 0.000 deg,	P = 30.000 deg,	R = 139.077 deg
};
P[311]{
   GP1:
	UF : 0, UT : 1,		CONFIG : 'N U T, 0, 0, 0',
	X = 1147.096  mm,	Y = 202.489  mm,	Z = -248.541  mm,
	W = 0.000 deg,	P = 30.000 deg,	R = 149.840 deg
};
P[312]{
   GP1:
	UF : 0, UT : 1,		CONFIG : 'N U T, 0, 0, 0',
	X = 1149.413  mm,	Y = 204.511  mm,	Z = -249.290  mm,
	W = 0.000 deg,	P = 30.000 deg,	R = 160.521 deg
};
P[313]{
   GP1:
	UF : 0, UT : 1,		CONFIG : 'N U T, 0, 0, 0',
	X = 1151.591  mm,	Y = 206.522  mm,	Z = -249.976  mm,
	W = 0.000 deg,	P = 30.000 deg,	R = 170.843 deg
};
P[314]{
   GP1:
	UF : 0, UT : 1,		CONFIG : 'N U T, 0, 0, 0',
	X = 1153.825  mm,	Y = 208.537  mm,	Z = -250.672  mm,
	W = 0.000 deg,	P = 30.000 deg,	R = 170.843 deg
};
P[315]{
   GP1:
	UF : 0, UT : 1,		CONFIG : 'N U T, 0, 0, 0',
	X = 1155.975  mm,	Y = 210.609  mm,	Z = -251.313  mm,
	W = 0.000 deg,	P = 30.000 deg,	R = 170.843 deg
};
P[316]{
   GP1:
	UF : 0, UT : 1,		CONFIG : 'N U T, 0, 0, 0',
	X = 1157.858  mm,	Y = 212.707  mm,	Z = -251.862  mm,
	W = 0.000 deg,	P = 30.000 deg,	R = 170.843 deg
};
P[317]{
   GP1:
	UF : 0, UT : 1,		CONFIG : 'N U T, 0, 0, 0',
	X = 1159.550  mm,	Y = 214.828  mm,	Z = -252.336  mm,
	W = 0.000 deg,	P = 30.000 deg,	R = 170.843 deg
};
P[318]{
   GP1:
	UF : 0, UT : 1,		CONFIG : 'N U T, 0, 0, 0',
	X = 1160.952  mm,	Y = 216.992  mm,	Z = -252.714  mm,
	W = 0.000 deg,	P = 30.000 deg,	R = 170.843 deg
};
P[319]{
   GP1:
	UF : 0, UT : 1,		CONFIG : 'N U T, 0, 0, 0',
	X = 1162.086  mm,	Y = 219.176  mm,	Z = -253.007  mm,
	W = 0.000 deg,	P = 30.000 deg,	R = 170.843 deg
};
P[320]{
   GP1:
	UF : 0, UT : 1,		CONFIG : 'N U T, 0, 0, 0',
	X = 1162.952  mm,	Y = 221.434  mm,	Z = -253.218  mm,
	W = 0.000 deg,	P = 30.000 deg,	R = 170.843 deg
};
P[321]{
   GP1:
	UF : 0, UT : 1,		CONFIG : 'N U T, 0, 0, 0',
	X = 1163.415  mm,	Y = 223.662  mm,	Z = -253.316  mm,
	W = 0.000 deg,	P = 30.000 deg,	R = 170.843 deg
};
P[322]{
   GP1:
	UF : 0, UT : 1,		CONFIG : 'N U T, 0, 0, 0',
	X = 1159.731  mm,	Y = 226.211  mm,	Z = -253.376  mm,
	W = 0.000 deg,	P = 30.000 deg,	R = 170.843 deg
};
P[323]{
   GP1:
	UF : 0, UT : 1,		CONFIG : 'N U T, 0, 0, 0',
	X = 1159.871  mm,	Y = 228.087  mm,	Z = -253.394  mm,
	W = 0.000 deg,	P = 30.000 deg,	R = 170.843 deg
};
P[324]{
   GP1:
	UF : 0, UT : 1,		CONFIG : 'N U T, 0, 0, 0',
	X = 1159.894  mm,	Y = 230.009  mm,	Z = -253.386  mm,
	W = 0.000 deg,	P = 30.000 deg,	R = 170.843 deg
};
P[325]{
   GP1:
	UF : 0, UT : 1,		CONFIG : 'N U T, 0, 0, 0',
	X = 1159.888  mm,	Y = 231.987  mm,	Z = -253.375  mm,
	W = 0.000 deg,	P = 30.000 deg,	R = 170.843 deg
};
P[326]{
   GP1:
	UF : 0, UT : 1,		CONFIG : 'N U T, 0, 0, 0',
	X = 1159.867  mm,	Y = 233.977  mm,	Z = -253.358  mm,
	W = 0.000 deg,	P = 30.000 deg,	R = 170.843 deg
};
P[327]{
   GP1:
	UF : 0, UT : 1,		CONFIG : 'N U T, 0, 0, 0',
	X = 1159.842  mm,	Y = 235.973  mm,	Z = -253.334  mm,
	W = 0.000 deg,	P = 30.000 deg,	R = 170.843 deg
};
P[328]{
   GP1:
	UF : 0, UT : 1,		CONFIG : 'N U T, 0, 0, 0',
	X = 1159.814  mm,	Y = 237.971  mm,	Z = -253.300  mm,
	W = 0.000 deg,	P = 30.000 deg,	R = 170.843 deg
};
P[329]{
   GP1:
	UF : 0, UT : 1,		CONFIG : 'N U T, 0, 0, 0',
	X = 1159.784  mm,	Y = 239.968  mm,	Z = -253.266  mm,
	W = 0.000 deg,	P = 30.000 deg,	R = 170.843 deg
};
P[330]{
   GP1:
	UF : 0, UT : 1,		CONFIG : 'N U T, 0, 0, 0',
	X = 1159.751  mm,	Y = 241.965  mm,	Z = -253.229  mm,
	W = 0.000 deg,	P = 30.000 deg,	R = 170.843 deg
};
P[331]{
   GP1:
	UF : 0, UT : 1,		CONFIG : 'N U T, 0, 0, 0',
	X = 1159.714  mm,	Y = 243.966  mm,	Z = -253.189  mm,
	W = 0.000 deg,	P = 30.000 deg,	R = 170.843 deg
};
P[332]{
   GP1:
	UF : 0, UT : 1,		CONFIG : 'N U T, 0, 0, 0',
	X = 1159.683  mm,	Y = 245.967  mm,	Z = -253.147  mm,
	W = 0.000 deg,	P = 30.000 deg,	R = 170.843 deg
};
P[333]{
   GP1:
	UF : 0, UT : 1,		CONFIG : 'N U T, 0, 0, 0',
	X = 1159.648  mm,	Y = 247.958  mm,	Z = -253.105  mm,
	W = 0.000 deg,	P = 30.000 deg,	R = 170.843 deg
};
P[334]{
   GP1:
	UF : 0, UT : 1,		CONFIG : 'N U T, 0, 0, 0',
	X = 1159.599  mm,	Y = 249.950  mm,	Z = -253.062  mm,
	W = 0.000 deg,	P = 30.000 deg,	R = 170.843 deg
};
P[335]{
   GP1:
	UF : 0, UT : 1,		CONFIG : 'N U T, 0, 0, 0',
	X = 1159.547  mm,	Y = 251.948  mm,	Z = -253.030  mm,
	W = 0.000 deg,	P = 30.000 deg,	R = 170.843 deg
};
P[336]{
   GP1:
	UF : 0, UT : 1,		CONFIG : 'N U T, 0, 0, 0',
	X = 1159.495  mm,	Y = 253.948  mm,	Z = -253.001  mm,
	W = 0.000 deg,	P = 30.000 deg,	R = 170.843 deg
};
/END
